 FB 13
BEGIN
   EN_R := TRUE;
   ID := W#16#16;
   R_ID := DW#16#16;
   NDR := FALSE;
   ERROR := FALSE;
   STATUS := W#16#0;
   RD_1 := P#DB28.DBX 0.0 BYTE 10;
   LEN := W#16#0;
   FB_ZUSTAND := B#16#0;
   EN_R_SAVE := FALSE;
   ID_SAVE := W#16#0;
   R_ID_SAVE := DW#16#0;
   FC_DATA_LEN := W#16#0;
   SD_1_SAVE0 := W#16#0;
   SD_1_SAVE2 := W#16#0;
   SD_1_SAVE4 := W#16#0;
   SD_1_SAVE6 := W#16#0;
   SD_1_SAVE8 := W#16#0;
   HS_REQ_BYTE.rii := FALSE;
   HS_REQ_BYTE.nva := FALSE;
   HS_REQ_BYTE.ofs := FALSE;
   HS_REQ_BYTE.dir := FALSE;
   HS_REQ_BYTE.res := FALSE;
   HS_REQ_BYTE.roc := FALSE;
   HS_REQ_BYTE.nls := FALSE;
   HS_REQ_BYTE.rlo := FALSE;
   HS_RESP_BYTE.aii := FALSE;
   HS_RESP_BYTE.sns := FALSE;
   HS_RESP_BYTE.sqc := FALSE;
   HS_RESP_BYTE.ads := FALSE;
   HS_RESP_BYTE.aoc := FALSE;
   HS_RESP_BYTE.rs1 := FALSE;
   HS_RESP_BYTE.cnr := FALSE;
   HS_RESP_BYTE.rs2 := FALSE;
   HS_RESP_DSNR := B#16#0;
   HS_RESP_OFFSET := W#16#0;
   SD_1_WORD0 := W#16#0;
   SD_1_COUNT := W#16#0;
   SD_1_DBNUMMER := W#16#0;
   SD_1_DWORD6 := DW#16#0;
   SD_1_TYP := B#16#0;
   SFC_PARAM.LEN := W#16#0;
   SFC_PARAM.DB_NUMMER := W#16#0;
   SFC_PARAM.START := DW#16#0;
   BUFFER[0] := W#16#0;
   BUFFER[1] := W#16#0;
   BUFFER[2] := W#16#0;
   BUFFER[3] := W#16#0;
   BUFFER[4] := W#16#0;
   BUFFER[5] := W#16#0;
   BUFFER[6] := W#16#0;
   BUFFER[7] := W#16#0;
   BUFFER[8] := W#16#0;
   BUFFER[9] := W#16#0;
   BUFFER[10] := W#16#0;
   BUFFER[11] := W#16#0;
   BUFFER[12] := W#16#0;
   BUFFER[13] := W#16#0;
   BUFFER[14] := W#16#0;
   BUFFER[15] := W#16#0;
   BUFFER[16] := W#16#0;
   BUFFER[17] := W#16#0;
   BUFFER[18] := W#16#0;
   BUFFER[19] := W#16#0;
   BUFFER[20] := W#16#0;
   BUFFER[21] := W#16#0;
   BUFFER[22] := W#16#0;
   BUFFER[23] := W#16#0;
   BUFFER[24] := W#16#0;
   BUFFER[25] := W#16#0;
   BUFFER[26] := W#16#0;
   BUFFER[27] := W#16#0;
   BUFFER[28] := W#16#0;
   BUFFER[29] := W#16#0;
   BUFFER[30] := W#16#0;
   BUFFER[31] := W#16#0;
   BUFFER[32] := W#16#0;
   BUFFER[33] := W#16#0;
   BUFFER[34] := W#16#0;
   BUFFER[35] := W#16#0;
   BUFFER[36] := W#16#0;
   BUFFER[37] := W#16#0;
   BUFFER[38] := W#16#0;
   BUFFER[39] := W#16#0;
   BUFFER[40] := W#16#0;
   BUFFER[41] := W#16#0;
   BUFFER[42] := W#16#0;
   BUFFER[43] := W#16#0;
   BUFFER[44] := W#16#0;
   BUFFER[45] := W#16#0;
   BUFFER[46] := W#16#0;
   BUFFER[47] := W#16#0;
   BUFFER[48] := W#16#0;
   BUFFER[49] := W#16#0;
   BUFFER[50] := W#16#0;
   BUFFER[51] := W#16#0;
   BUFFER[52] := W#16#0;
   BUFFER[53] := W#16#0;
   BUFFER[54] := W#16#0;
   BUFFER[55] := W#16#0;
   BUFFER[56] := W#16#0;
   BUFFER[57] := W#16#0;
   BUFFER[58] := W#16#0;
   BUFFER[59] := W#16#0;
   BUFFER[60] := W#16#0;
   BUFFER[61] := W#16#0;
   BUFFER[62] := W#16#0;
   BUFFER[63] := W#16#0;
   BUFFER[64] := W#16#0;
   BUFFER[65] := W#16#0;
   BUFFER[66] := W#16#0;
   BUFFER[67] := W#16#0;
   BUFFER[68] := W#16#0;
   BUFFER[69] := W#16#0;
   BUFFER[70] := W#16#0;
   BUFFER[71] := W#16#0;
   BUFFER[72] := W#16#0;
   BUFFER[73] := W#16#0;
   BUFFER[74] := W#16#0;
   BUFFER[75] := W#16#0;
   BUFFER[76] := W#16#0;
   BUFFER[77] := W#16#0;
   BUFFER[78] := W#16#0;
   BUFFER[79] := W#16#0;
   BUFFER[80] := W#16#0;
   BUFFER[81] := W#16#0;
   BUFFER[82] := W#16#0;
   BUFFER[83] := W#16#0;
   BUFFER[84] := W#16#0;
   BUFFER[85] := W#16#0;
   BUFFER[86] := W#16#0;
   BUFFER[87] := W#16#0;
   BUFFER[88] := W#16#0;
   BUFFER[89] := W#16#0;
   BUFFER[90] := W#16#0;
   BUFFER[91] := W#16#0;
   BUFFER[92] := W#16#0;
   BUFFER[93] := W#16#0;
   BUFFER[94] := W#16#0;
   BUFFER[95] := W#16#0;
   BUFFER[96] := W#16#0;
   BUFFER[97] := W#16#0;
   BUFFER[98] := W#16#0;
   BUFFER[99] := W#16#0;
   BUFFER[100] := W#16#0;
   BUFFER[101] := W#16#0;
   BUFFER[102] := W#16#0;
   BUFFER[103] := W#16#0;
   BUFFER[104] := W#16#0;
   BUFFER[105] := W#16#0;
   BUFFER[106] := W#16#0;
   BUFFER[107] := W#16#0;
   BUFFER[108] := W#16#0;
   BUFFER[109] := W#16#0;
   BUFFER[110] := W#16#0;
   BUFFER[111] := W#16#0;
   BUFFER[112] := W#16#0;
   BUFFER[113] := W#16#0;
   BUFFER[114] := W#16#0;
   BUFFER[115] := W#16#0;
   BUFFER[116] := W#16#0;
   BUFFER[117] := W#16#0;
   BUFFER[118] := W#16#0;
   BUFFER[119] := W#16#0;
   REASON_FOR_CLOSE := B#16#0;
   DS_NR := B#16#0;
   MAX_PUFF_LEN_SAVE := W#16#0;
   TYP_BOOL := FALSE;
   KANAL_PROBLEM := FALSE;
   KOMM_PROBLEM := FALSE;
   RECV_STARTED := FALSE;
   SEND_STARTED := FALSE;
   RESET_REQUEST := FALSE;
   RESET_EXECUTED := FALSE;
   DS200_BUSY := FALSE;
   LADDR_PTR := DW#16#0;
   LADDR := W#16#0;
   ZIEL_BYTE_SAVE := B#16#0;
   BOOL_ZIEL_BAD := FALSE;
   PARAM_OFFSET := DW#16#0;
   SLEEP := B#16#0;
   SLEEP_EXT := B#16#0;
   ID_CLOSE := W#16#0;
   RUNNING_LEN := W#16#0;
   FB_KENNUNG := B#16#F2;
   RESERVE := B#16#0;
   ZUSTAND_WEICHE := B#16#2;
   SFB_AUFRUF.EN_R := TRUE;
   SFB_AUFRUF.ID := W#16#16;
   SFB_AUFRUF.R_ID := DW#16#16;
   SFB_AUFRUF.NDR := FALSE;
   SFB_AUFRUF.ERROR := FALSE;
   SFB_AUFRUF.STATUS := W#16#0;
   SFB_AUFRUF.RD_1 := P#DB28.DBX 0.0 BYTE 10;
   SFB_AUFRUF.LEN := W#16#0;
   SFB_AUFRUF.INDEX := W#16#801;
   ZUSTAND_WEICHE_1 := B#16#CA;
END_DATA_BLOCK

DATA_BLOCK DB 326
TITLE =
AUTHOR : ICom
FAMILY : DIAGNOSE
VERSION : 0.0

 FB 327
BEGIN
   IN0 := 327;
   OUT1 := DW#16#0;
   STAT2[1] := B#16#0;
   STAT2[2] := B#16#64;
   STAT2[3] := B#16#1;
   STAT2[4] := B#16#10;
   STAT2[5] := B#16#F0;
   STAT2[6] := B#16#0;
   STAT2[7] := B#16#0;
   STAT2[8] := B#16#0;
   STAT2[9] := B#16#0;
   STAT2[10] := B#16#0;
   STAT2[11] := B#16#0;
   STAT2[12] := B#16#0;
   STAT2[13] := B#16#0;
   STAT2[14] := B#16#0;
   STAT2[15] := B#16#0;
   STAT2[16] := B#16#0;
   STAT2[17] := B#16#0;
   STAT2[18] := B#16#0;
   STAT2[19] := B#16#0;
   STAT2[20] := B#16#0;
   STAT2[21] := B#16#40;
   STAT2[22] := B#16#0;
   STAT2[23] := B#16#0;
   STAT2[24] := B#16#0;
   STAT2[25] := B#16#0;
   STAT2[26] := B#16#0;
   STAT2[27] := B#16#0;
   STAT2[28] := B#16#0;
   STAT2[29] := B#16#0;
   STAT2[30] := B#16#0;
   STAT2[31] := B#16#0;
   STAT2[32] := B#16#0;
   STAT2[33] := B#16#0;
   STAT2[34] := B#16#0;
   STAT2[35] := B#16#0;
   STAT2[36] := B#16#0;
   STAT2[37] := B#16#0;
   STAT2[38] := B#16#0;
   STAT2[39] := B#16#0;
   STAT2[40] := B#16#0;
   STAT2[41] := B#16#0;
   STAT2[42] := B#16#0;
   STAT2[43] := B#16#0;
   STAT2[44] := B#16#0;
   STAT2[45] := B#16#0;
   STAT2[46] := B#16#0;
   STAT2[47] := B#16#0;
   STAT2[48] := B#16#0;
   STAT2[49] := B#16#0;
   STAT2[50] := B#16#0;
   STAT2[51] := B#16#0;
   STAT2[52] := B#16#0;
   STAT2[53] := B#16#0;
   STAT2[54] := B#16#0;
   STAT2[55] := B#16#0;
   STAT2[56] := B#16#0;
   STAT2[57] := B#16#0;
   STAT2[58] := B#16#0;
   STAT2[59] := B#16#0;
   STAT2[60] := B#16#0;
   STAT2[61] := B#16#0;
   STAT2[62] := B#16#0;
   STAT2[63] := B#16#0;
   STAT2[64] := B#16#0;
   STAT2[65] := B#16#0;
   STAT2[66] := B#16#0;
   STAT2[67] := B#16#0;
   STAT2[68] := B#16#0;
   STAT2[69] := B#16#0;
   STAT2[70] := B#16#0;
   STAT2[71] := B#16#0;
   STAT2[72] := B#16#0;
   STAT2[73] := B#16#0;
   STAT2[74] := B#16#0;
   STAT2[75] := B#16#0;
   STAT2[76] := B#16#0;
   STAT2[77] := B#16#0;
   STAT2[78] := B#16#0;
   STAT2[79] := B#16#0;
   STAT2[80] := B#16#0;
   STAT2[81] := B#16#0;
   STAT2[82] := B#16#0;
   STAT2[83] := B#16#0;
   STAT2[84] := B#16#0;
   STAT2[85] := B#16#0;
   STAT2[86] := B#16#0;
   STAT2[87] := B#16#0;
   STAT2[88] := B#16#0;
   STAT2[89] := B#16#0;
   STAT2[90] := B#16#0;
   STAT2[91] := B#16#0;
   STAT2[92] := B#16#0;
   STAT2[93] := B#16#0;
   STAT2[94] := B#16#0;
   STAT2[95] := B#16#0;
   STAT2[96] := B#16#0;
   STAT2[97] := B#16#0;
   STAT2[98] := B#16#0;
   STAT2[99] := B#16#0;
   STAT2[100] := B#16#0;
   STAT2[101] := B#16#0;
   STAT2[102] := B#16#0;
   STAT2[103] := B#16#0;
   STAT2[104] := B#16#0;
   STAT2[105] := B#16#0;
   STAT2[106] := B#16#0;
   STAT2[107] := B#16#0;
   STAT2[108] := B#16#0;
   STAT2[109] := B#16#0;
   STAT2[110] := B#16#0;
   STAT2[111] := B#16#0;
   STAT2[112] := B#16#0;
   STAT2[113] := B#16#0;
   STAT2[114] := B#16#0;
   STAT2[115] := B#16#0;
   STAT2[116] := B#16#0;
   STAT2[117] := B#16#0;
   STAT2[118] := B#16#0;
   STAT2[119] := B#16#0;
   STAT2[120] := B#16#0;
   STAT2[121] := B#16#0;
   STAT2[122] := B#16#0;
   STAT2[123] := B#16#0;
   STAT2[124] := B#16#0;
   STAT2[125] := B#16#0;
   STAT2[126] := B#16#0;
   STAT2[127] := B#16#0;
   STAT2[128] := B#16#0;
   STAT2[129] := B#16#0;
   STAT2[130] := B#16#0;
   STAT2[131] := B#16#0;
   STAT2[132] := B#16#0;
   STAT2[133] := B#16#0;
   STAT2[134] := B#16#0;
   STAT2[135] := B#16#0;
   STAT2[136] := B#16#0;
   STAT2[137] := B#16#0;
   STAT2[138] := B#16#0;
   STAT2[139] := B#16#0;
   STAT2[140] := B#16#0;
   STAT2[141] := B#16#0;
   STAT2[142] := B#16#0;
   STAT2[143] := B#16#0;
   STAT2[144] := B#16#0;
   STAT2[145] := B#16#0;
   STAT2[146] := B#16#0;
   STAT2[147] := B#16#0;
   STAT2[148] := B#16#0;
   STAT2[149] := B#16#0;
   STAT2[150] := B#16#0;
   STAT2[151] := B#16#0;
   STAT2[152] := B#16#0;
   STAT2[153] := B#16#0;
   STAT2[154] := B#16#0;
   STAT2[155] := B#16#0;
   STAT2[156] := B#16#0;
   STAT2[157] := B#16#0;
   STAT2[158] := B#16#0;
   STAT2[159] := B#16#0;
   STAT2[160] := B#16#0;
   STAT2[161] := B#16#0;
   STAT2[162] := B#16#0;
   STAT2[163] := B#16#0;
   STAT2[164] := B#16#0;
   STAT2[165] := B#16#0;
   STAT2[166] := B#16#0;
   STAT2[167] := B#16#0;
   STAT2[168] := B#16#0;
   STAT2[169] := B#16#0;
   STAT2[170] := B#16#0;
   STAT2[171] := B#16#0;
   STAT2[172] := B#16#0;
   STAT2[173] := B#16#0;
   STAT2[174] := B#16#0;
   STAT2[175] := B#16#0;
   STAT2[176] := B#16#0;
   STAT2[177] := B#16#0;
   STAT2[178] := B#16#0;
   STAT2[179] := B#16#0;
   STAT2[180] := B#16#0;
   STAT2[181] := B#16#0;
   STAT2[182] := B#16#0;
   STAT2[183] := B#16#0;
   STAT2[184] := B#16#0;
   STAT2[185] := B#16#0;
   STAT2[186] := B#16#0;
   STAT2[187] := B#16#0;
   STAT2[188] := B#16#0;
   STAT2[189] := B#16#0;
   STAT2[190] := B#16#0;
   STAT2[191] := B#16#0;
   STAT2[192] := B#16#0;
   STAT2[193] := B#16#0;
   STAT2[194] := B#16#0;
   STAT2[195] := B#16#0;
   STAT2[196] := B#16#0;
   STAT2[197] := B#16#0;
   STAT2[198] := B#16#0;
   STAT2[199] := B#16#0;
   STAT2[200] := B#16#0;
   STAT2[201] := B#16#0;
   STAT2[202] := B#16#0;
   STAT2[203] := B#16#0;
   STAT2[204] := B#16#0;
   STAT2[205] := B#16#0;
   STAT2[206] := B#16#0;
   STAT2[207] := B#16#0;
   STAT2[208] := B#16#0;
   STAT2[209] := B#16#0;
   STAT2[210] := B#16#0;
   STAT2[211] := B#16#0;
   STAT2[212] := B#16#0;
   STAT2[213] := B#16#0;
   STAT2[214] := B#16#0;
   STAT2[215] := B#16#0;
   STAT2[216] := B#16#0;
   STAT2[217] := B#16#0;
   STAT2[218] := B#16#0;
   STAT2[219] := B#16#0;
   STAT2[220] := B#16#0;
   STAT2[221] := B#16#0;
   STAT2[222] := B#16#0;
   STAT2[223] := B#16#0;
   STAT2[224] := B#16#0;
   STAT2[225] := B#16#0;
   STAT2[226] := B#16#0;
   STAT2[227] := B#16#0;
   STAT2[228] := B#16#0;
   STAT2[229] := B#16#0;
   STAT2[230] := B#16#0;
   STAT2[231] := B#16#0;
   STAT2[232] := B#16#0;
   STAT2[233] := B#16#0;
   STAT2[234] := B#16#0;
   STAT2[235] := B#16#0;
   STAT2[236] := B#16#0;
   STAT2[237] := B#16#0;
   STAT2[238] := B#16#0;
   STAT2[239] := B#16#0;
   STAT2[240] := B#16#0;
   STAT2[241] := B#16#0;
   STAT2[242] := B#16#0;
   STAT2[243] := B#16#0;
   STAT2[244] := B#16#0;
   STAT2[245] := B#16#0;
   STAT2[246] := B#16#0;
   STAT2[247] := B#16#0;
   STAT2[248] := B#16#0;
   STAT2[249] := B#16#0;
   STAT2[250] := B#16#0;
   STAT2[251] := B#16#0;
   STAT2[252] := B#16#0;
   STAT2[253] := B#16#0;
   STAT2[254] := B#16#0;
   STAT2[255] := B#16#0;
   STAT2[256] := B#16#0;
   STAT2[257] := B#16#0;
   STAT2[258] := B#16#0;
   STAT2[259] := B#16#0;
   STAT2[260] := B#16#64;
   STAT2[261] := B#16#1;
   STAT2[262] := B#16#10;
   STAT2[263] := B#16#F0;
   STAT2[264] := B#16#0;
   STAT2[265] := B#16#0;
   STAT2[266] := B#16#0;
   STAT2[267] := B#16#0;
   STAT2[268] := B#16#0;
   STAT2[269] := B#16#0;
   STAT2[270] := B#16#0;
   STAT2[271] := B#16#0;
   STAT2[272] := B#16#0;
   STAT2[273] := B#16#0;
   STAT2[274] := B#16#0;
   STAT2[275] := B#16#0;
   STAT2[276] := B#16#0;
   STAT2[277] := B#16#0;
   STAT2[278] := B#16#0;
   STAT2[279] := B#16#40;
   STAT2[280] := B#16#0;
   STAT2[281] := B#16#0;
   STAT2[282] := B#16#0;
   STAT2[283] := B#16#0;
   STAT2[284] := B#16#0;
   STAT2[285] := B#16#0;
   STAT2[286] := B#16#0;
   STAT2[287] := B#16#0;
   STAT2[288] := B#16#0;
   STAT2[289] := B#16#0;
   STAT2[290] := B#16#0;
   STAT2[291] := B#16#0;
   STAT2[292] := B#16#0;
   STAT2[293] := B#16#0;
   STAT2[294] := B#16#0;
   STAT2[295] := B#16#0;
   STAT2[296] := B#16#0;
   STAT2[297] := B#16#0;
   STAT2[298] := B#16#0;
   STAT2[299] := B#16#0;
   STAT2[300] := B#16#0;
   STAT2[301] := B#16#0;
   STAT2[302] := B#16#0;
   STAT2[303] := B#16#0;
   STAT2[304] := B#16#0;
   STAT2[305] := B#16#0;
   STAT2[306] := B#16#0;
   STAT2[307] := B#16#0;
   STAT2[308] := B#16#0;
   STAT2[309] := B#16#0;
   STAT2[310] := B#16#0;
   STAT2[311] := B#16#0;
   STAT2[312] := B#16#0;
   STAT2[313] := B#16#0;
   STAT2[314] := B#16#0;
   STAT2[315] := B#16#0;
   STAT2[316] := B#16#0;
   STAT2[317] := B#16#0;
   STAT2[318] := B#16#0;
   STAT2[319] := B#16#0;
   STAT2[320] := B#16#0;
   STAT2[321] := B#16#0;
   STAT2[322] := B#16#0;
   STAT2[323] := B#16#0;
   STAT2[324] := B#16#0;
   STAT2[325] := B#16#0;
   STAT2[326] := B#16#0;
   STAT2[327] := B#16#0;
   STAT2[328] := B#16#0;
   STAT2[329] := B#16#0;
   STAT2[330] := B#16#0;
   STAT2[331] := B#16#0;
   STAT2[332] := B#16#0;
   STAT2[333] := B#16#0;
   STAT2[334] := B#16#0;
   STAT2[335] := B#16#0;
   STAT2[336] := B#16#0;
   STAT2[337] := B#16#0;
   STAT2[338] := B#16#0;
   STAT2[339] := B#16#0;
   STAT2[340] := B#16#0;
   STAT2[341] := B#16#0;
   STAT2[342] := B#16#0;
   STAT2[343] := B#16#0;
   STAT2[344] := B#16#0;
   STAT2[345] := B#16#0;
   STAT2[346] := B#16#0;
   STAT2[347] := B#16#0;
   STAT2[348] := B#16#0;
   STAT2[349] := B#16#0;
   STAT2[350] := B#16#0;
   STAT2[351] := B#16#0;
   STAT2[352] := B#16#0;
   STAT2[353] := B#16#0;
   STAT2[354] := B#16#0;
   STAT2[355] := B#16#0;
   STAT2[356] := B#16#0;
   STAT2[357] := B#16#0;
   STAT2[358] := B#16#0;
   STAT2[359] := B#16#0;
   STAT2[360] := B#16#0;
   STAT2[361] := B#16#0;
   STAT2[362] := B#16#0;
   STAT2[363] := B#16#0;
   STAT2[364] := B#16#0;
   STAT2[365] := B#16#0;
   STAT2[366] := B#16#0;
   STAT2[367] := B#16#0;
   STAT2[368] := B#16#0;
   STAT2[369] := B#16#0;
   STAT2[370] := B#16#0;
   STAT2[371] := B#16#0;
   STAT2[372] := B#16#0;
   STAT2[373] := B#16#0;
   STAT2[374] := B#16#0;
   STAT2[375] := B#16#0;
   STAT2[376] := B#16#0;
   STAT2[377] := B#16#0;
   STAT2[378] := B#16#0;
   STAT2[379] := B#16#0;
   STAT2[380] := B#16#0;
   STAT2[381] := B#16#0;
   STAT2[382] := B#16#0;
   STAT2[383] := B#16#0;
   STAT2[384] := B#16#0;
   STAT2[385] := B#16#0;
   STAT2[386] := B#16#0;
   STAT2[387] := B#16#0;
   STAT2[388] := B#16#0;
   STAT2[389] := B#16#0;
   STAT2[390] := B#16#0;
   STAT2[391] := B#16#0;
   STAT2[392] := B#16#0;
   STAT2[393] := B#16#0;
   STAT2[394] := B#16#0;
   STAT2[395] := B#16#0;
   STAT2[396] := B#16#0;
   STAT2[397] := B#16#0;
   STAT2[398] := B#16#0;
   STAT2[399] := B#16#0;
   STAT2[400] := B#16#0;
   STAT2[401] := B#16#0;
   STAT2[402] := B#16#0;
   STAT2[403] := B#16#0;
   STAT2[404] := B#16#0;
   STAT2[405] := B#16#0;
   STAT2[406] := B#16#0;
   STAT2[407] := B#16#0;
   STAT2[408] := B#16#0;
   STAT2[409] := B#16#0;
   STAT2[410] := B#16#0;
   STAT2[411] := B#16#0;
   STAT2[412] := B#16#0;
   STAT2[413] := B#16#0;
   STAT2[414] := B#16#0;
   STAT2[415] := B#16#0;
   STAT2[416] := B#16#0;
   STAT2[417] := B#16#0;
   STAT2[418] := B#16#0;
   STAT2[419] := B#16#0;
   STAT2[420] := B#16#0;
   STAT2[421] := B#16#0;
   STAT2[422] := B#16#0;
   STAT2[423] := B#16#0;
   STAT2[424] := B#16#0;
   STAT2[425] := B#16#0;
   STAT2[426] := B#16#0;
   STAT2[427] := B#16#0;
   STAT2[428] := B#16#0;
   STAT2[429] := B#16#0;
   STAT2[430] := B#16#0;
   STAT2[431] := B#16#0;
   STAT2[432] := B#16#0;
   STAT2[433] := B#16#0;
   STAT2[434] := B#16#0;
   STAT2[435] := B#16#0;
   STAT2[436] := B#16#0;
   STAT2[437] := B#16#0;
   STAT2[438] := B#16#0;
   STAT2[439] := B#16#0;
   STAT2[440] := B#16#0;
   STAT2[441] := B#16#0;
   STAT2[442] := B#16#0;
   STAT2[443] := B#16#0;
   STAT2[444] := B#16#0;
   STAT2[445] := B#16#0;
   STAT2[446] := B#16#0;
   STAT2[447] := B#16#0;
   STAT2[448] := B#16#0;
   STAT2[449] := B#16#0;
   STAT2[450] := B#16#0;
   STAT2[451] := B#16#0;
   STAT2[452] := B#16#0;
   STAT2[453] := B#16#0;
   STAT2[454] := B#16#0;
   STAT2[455] := B#16#0;
   STAT2[456] := B#16#0;
   STAT2[457] := B#16#0;
   STAT2[458] := B#16#0;
   STAT2[459] := B#16#0;
   STAT2[460] := B#16#0;
   STAT2[461] := B#16#0;
   STAT2[462] := B#16#0;
   STAT2[463] := B#16#0;
   STAT2[464] := B#16#0;
   STAT2[465] := B#16#0;
   STAT2[466] := B#16#0;
   STAT2[467] := B#16#0;
   STAT2[468] := B#16#0;
   STAT2[469] := B#16#0;
   STAT2[470] := B#16#0;
   STAT2[471] := B#16#0;
   STAT2[472] := B#16#0;
   STAT2[473] := B#16#0;
   STAT2[474] := B#16#0;
   STAT2[475] := B#16#0;
   STAT2[476] := B#16#0;
   STAT2[477] := B#16#0;
   STAT2[478] := B#16#0;
   STAT2[479] := B#16#0;
   STAT2[480] := B#16#0;
   STAT2[481] := B#16#0;
   STAT2[482] := B#16#0;
   STAT2[483] := B#16#0;
   STAT2[484] := B#16#0;
   STAT2[485] := B#16#0;
   STAT2[486] := B#16#0;
   STAT2[487] := B#16#0;
   STAT2[488] := B#16#0;
   STAT2[489] := B#16#0;
   STAT2[490] := B#16#0;
   STAT2[491] := B#16#0;
   STAT2[492] := B#16#0;
   STAT2[493] := B#16#0;
   STAT2[494] := B#16#0;
   STAT2[495] := B#16#0;
   STAT2[496] := B#16#0;
   STAT2[497] := B#16#0;
   STAT2[498] := B#16#0;
   STAT2[499] := B#16#0;
   STAT2[500] := B#16#0;
   STAT2[501] := B#16#0;
   STAT2[502] := B#16#0;
   STAT2[503] := B#16#0;
   STAT2[504] := B#16#0;
   STAT2[505] := B#16#0;
   STAT2[506] := B#16#0;
   STAT2[507] := B#16#0;
   STAT2[508] := B#16#0;
   STAT2[509] := B#16#0;
   STAT2[510] := B#16#0;
   STAT2[511] := B#16#0;
   STAT2[512] := B#16#0;
   STAT2[513] := B#16#0;
   STAT2[514] := B#16#0;
   STAT2[515] := B#16#0;
   STAT2[516] := B#16#0;
   STAT2[517] := B#16#0;
   STAT2[518] := B#16#64;
   STAT2[519] := B#16#0;
   STAT2[520] := B#16#0;
   STAT2[521] := B#16#0;
   STAT2[522] := B#16#0;
   STAT2[523] := B#16#0;
   STAT2[524] := B#16#0;
   STAT2[525] := B#16#0;
   STAT2[526] := B#16#0;
   STAT2[527] := B#16#0;
   STAT2[528] := B#16#0;
   STAT2[529] := B#16#0;
   STAT2[530] := B#16#0;
   STAT2[531] := B#16#0;
   STAT2[532] := B#16#0;
   STAT2[533] := B#16#0;
   STAT2[534] := B#16#0;
   STAT2[535] := B#16#0;
   STAT2[536] := B#16#0;
   STAT2[537] := B#16#0;
   STAT2[538] := B#16#0;
   STAT2[539] := B#16#0;
   STAT2[540] := B#16#0;
   STAT2[541] := B#16#0;
   STAT2[542] := B#16#0;
   STAT2[543] := B#16#0;
   STAT2[544] := B#16#0;
   STAT2[545] := B#16#0;
   STAT2[546] := B#16#0;
   STAT2[547] := B#16#0;
   STAT2[548] := B#16#0;
   STAT2[549] := B#16#0;
   STAT2[550] := B#16#0;
   STAT2[551] := B#16#0;
   STAT2[552] := B#16#0;
   STAT2[553] := B#16#0;
   STAT2[554] := B#16#0;
   STAT2[555] := B#16#0;
   STAT2[556] := B#16#0;
   STAT2[557] := B#16#0;
   STAT2[558] := B#16#0;
   STAT2[559] := B#16#0;
   STAT2[560] := B#16#0;
   STAT2[561] := B#16#0;
   STAT2[562] := B#16#0;
   STAT2[563] := B#16#0;
   STAT2[564] := B#16#0;
   STAT2[565] := B#16#0;
   STAT2[566] := B#16#0;
   STAT2[567] := B#16#0;
   STAT2[568] := B#16#0;
   STAT2[569] := B#16#0;
   STAT2[570] := B#16#0;
   STAT2[571] := B#16#0;
   STAT2[572] := B#16#0;
   STAT2[573] := B#16#0;
   STAT2[574] := B#16#0;
   STAT2[575] := B#16#0;
   STAT2[576] := B#16#0;
   STAT2[577] := B#16#0;
   STAT2[578] := B#16#0;
   STAT2[579] := B#16#0;
   STAT2[580] := B#16#0;
   STAT2[581] := B#16#0;
   STAT2[582] := B#16#0;
   STAT2[583] := B#16#0;
   STAT2[584] := B#16#0;
   STAT2[585] := B#16#0;
   STAT2[586] := B#16#0;
   STAT2[587] := B#16#0;
   STAT2[588] := B#16#0;
   STAT2[589] := B#16#0;
   STAT2[590] := B#16#0;
   STAT2[591] := B#16#0;
   STAT2[592] := B#16#0;
   STAT2[593] := B#16#0;
   STAT2[594] := B#16#0;
   STAT2[595] := B#16#0;
   STAT2[596] := B#16#0;
   STAT2[597] := B#16#0;
   STAT2[598] := B#16#0;
   STAT2[599] := B#16#0;
   STAT2[600] := B#16#0;
   STAT2[601] := B#16#0;
   STAT2[602] := B#16#0;
   STAT2[603] := B#16#0;
   STAT2[604] := B#16#0;
   STAT2[605] := B#16#0;
   STAT2[606] := B#16#0;
   STAT2[607] := B#16#0;
   STAT2[608] := B#16#0;
   STAT2[609] := B#16#0;
   STAT2[610] := B#16#0;
   STAT2[611] := B#16#0;
   STAT2[612] := B#16#0;
   STAT2[613] := B#16#0;
   STAT2[614] := B#16#0;
   STAT2[615] := B#16#0;
   STAT2[616] := B#16#0;
   STAT2[617] := B#16#0;
   STAT2[618] := B#16#0;
   STAT2[619] := B#16#0;
   STAT2[620] := B#16#0;
   STAT2[621] := B#16#0;
   STAT2[622] := B#16#0;
   STAT2[623] := B#16#0;
   STAT2[624] := B#16#0;
   STAT2[625] := B#16#0;
   STAT2[626] := B#16#0;
   STAT2[627] := B#16#0;
   STAT2[628] := B#16#0;
   STAT2[629] := B#16#0;
   STAT2[630] := B#16#0;
   STAT2[631] := B#16#0;
   STAT2[632] := B#16#0;
   STAT2[633] := B#16#0;
   STAT2[634] := B#16#0;
   STAT2[635] := B#16#0;
   STAT2[636] := B#16#0;
   STAT2[637] := B#16#0;
   STAT2[638] := B#16#0;
   STAT2[639] := B#16#0;
   STAT2[640] := B#16#0;
   STAT2[641] := B#16#0;
   STAT2[642] := B#16#0;
   STAT2[643] := B#16#0;
   STAT2[644] := B#16#0;
   STAT2[645] := B#16#0;
   STAT2[646] := B#16#0;
   STAT2[647] := B#16#0;
   STAT2[648] := B#16#0;
   STAT2[649] := B#16#0;
   STAT2[650] := B#16#0;
   STAT2[651] := B#16#0;
   STAT2[652] := B#16#0;
   STAT2[653] := B#16#0;
   STAT2[654] := B#16#0;
   STAT2[655] := B#16#0;
   STAT2[656] := B#16#0;
   STAT2[657] := B#16#0;
   STAT2[658] := B#16#0;
   STAT2[659] := B#16#0;
   STAT2[660] := B#16#0;
   STAT2[661] := B#16#0;
   STAT2[662] := B#16#0;
   STAT2[663] := B#16#0;
   STAT2[664] := B#16#0;
   STAT2[665] := B#16#0;
   STAT2[666] := B#16#0;
   STAT2[667] := B#16#0;
   STAT2[668] := B#16#0;
   STAT2[669] := B#16#0;
   STAT2[670] := B#16#0;
   STAT2[671] := B#16#0;
   STAT2[672] := B#16#0;
   STAT2[673] := B#16#0;
   STAT2[674] := B#16#0;
   STAT2[675] := B#16#0;
   STAT2[676] := B#16#0;
   STAT2[677] := B#16#0;
   STAT2[678] := B#16#0;
   STAT2[679] := B#16#0;
   STAT2[680] := B#16#0;
   STAT2[681] := B#16#0;
   STAT2[682] := B#16#0;
   STAT2[683] := B#16#0;
   STAT2[684] := B#16#0;
   STAT2[685] := B#16#0;
   STAT2[686] := B#16#0;
   STAT2[687] := B#16#0;
   STAT2[688] := B#16#0;
   STAT2[689] := B#16#0;
   STAT2[690] := B#16#0;
   STAT2[691] := B#16#0;
   STAT2[692] := B#16#0;
   STAT2[693] := B#16#0;
   STAT2[694] := B#16#0;
   STAT2[695] := B#16#0;
   STAT2[696] := B#16#0;
   STAT2[697] := B#16#0;
   STAT2[698] := B#16#0;
   STAT2[699] := B#16#0;
   STAT2[700] := B#16#0;
   STAT2[701] := B#16#0;
   STAT2[702] := B#16#0;
   STAT2[703] := B#16#0;
   STAT2[704] := B#16#0;
   STAT2[705] := B#16#0;
   STAT2[706] := B#16#0;
   STAT2[707] := B#16#0;
   STAT2[708] := B#16#0;
   STAT2[709] := B#16#0;
   STAT2[710] := B#16#0;
   STAT2[711] := B#16#0;
   STAT2[712] := B#16#0;
   STAT2[713] := B#16#0;
   STAT2[714] := B#16#0;
   STAT2[715] := B#16#0;
   STAT2[716] := B#16#0;
   STAT2[717] := B#16#0;
   STAT2[718] := B#16#0;
   STAT2[719] := B#16#0;
   STAT2[720] := B#16#0;
   STAT2[721] := B#16#0;
   STAT2[722] := B#16#0;
   STAT2[723] := B#16#0;
   STAT2[724] := B#16#0;
   STAT2[725] := B#16#0;
   STAT2[726] := B#16#0;
   STAT2[727] := B#16#0;
   STAT2[728] := B#16#0;
   STAT2[729] := B#16#0;
   STAT2[730] := B#16#0;
   STAT2[731] := B#16#0;
   STAT2[732] := B#16#0;
   STAT2[733] := B#16#0;
   STAT2[734] := B#16#0;
   STAT2[735] := B#16#0;
   STAT2[736] := B#16#0;
   STAT2[737] := B#16#0;
   STAT2[738] := B#16#0;
   STAT2[739] := B#16#0;
   STAT2[740] := B#16#0;
   STAT2[741] := B#16#0;
   STAT2[742] := B#16#0;
   STAT2[743] := B#16#0;
   STAT2[744] := B#16#0;
   STAT2[745] := B#16#0;
   STAT2[746] := B#16#0;
   STAT2[747] := B#16#0;
   STAT2[748] := B#16#0;
   STAT2[749] := B#16#0;
   STAT2[750] := B#16#0;
   STAT2[751] := B#16#0;
   STAT2[752] := B#16#0;
   STAT2[753] := B#16#0;
   STAT2[754] := B#16#0;
   STAT2[755] := B#16#0;
   STAT2[756] := B#16#0;
   STAT2[757] := B#16#0;
   STAT2[758] := B#16#0;
   STAT2[759] := B#16#0;
   STAT2[760] := B#16#0;
   STAT2[761] := B#16#0;
   STAT2[762] := B#16#0;
   STAT2[763] := B#16#0;
   STAT2[764] := B#16#0;
   STAT2[765] := B#16#0;
   STAT2[766] := B#16#0;
   STAT2[767] := B#16#0;
   STAT2[768] := B#16#0;
   STAT2[769] := B#16#0;
   STAT2[770] := B#16#0;
   STAT2[771] := B#16#0;
   STAT2[772] := B#16#0;
   STAT2[773] := B#16#0;
   STAT2[774] := B#16#0;
   STAT2[775] := B#16#0;
   STAT2[776] := B#16#64;
   STAT2[777] := B#16#0;
   STAT2[778] := B#16#0;
   STAT2[779] := B#16#0;
   STAT2[780] := B#16#0;
   STAT2[781] := B#16#0;
   STAT2[782] := B#16#0;
   STAT2[783] := B#16#0;
   STAT2[784] := B#16#0;
   STAT2[785] := B#16#0;
   STAT2[786] := B#16#0;
   STAT2[787] := B#16#0;
   STAT2[788] := B#16#0;
   STAT2[789] := B#16#0;
   STAT2[790] := B#16#0;
   STAT2[791] := B#16#0;
   STAT2[792] := B#16#0;
   STAT2[793] := B#16#0;
   STAT2[794] := B#16#0;
   STAT2[795] := B#16#0;
   STAT2[796] := B#16#0;
   STAT2[797] := B#16#0;
   STAT2[798] := B#16#0;
   STAT2[799] := B#16#0;
   STAT2[800] := B#16#0;
   STAT2[801] := B#16#0;
   STAT2[802] := B#16#0;
   STAT2[803] := B#16#0;
   STAT2[804] := B#16#0;
   STAT2[805] := B#16#0;
   STAT2[806] := B#16#0;
   STAT2[807] := B#16#0;
   STAT2[808] := B#16#0;
   STAT2[809] := B#16#0;
   STAT2[810] := B#16#0;
   STAT2[811] := B#16#0;
   STAT2[812] := B#16#0;
   STAT2[813] := B#16#0;
   STAT2[814] := B#16#0;
   STAT2[815] := B#16#0;
   STAT2[816] := B#16#0;
   STAT2[817] := B#16#0;
   STAT2[818] := B#16#0;
   STAT2[819] := B#16#0;
   STAT2[820] := B#16#0;
   STAT2[821] := B#16#0;
   STAT2[822] := B#16#0;
   STAT2[823] := B#16#0;
   STAT2[824] := B#16#0;
   STAT2[825] := B#16#0;
   STAT2[826] := B#16#0;
   STAT2[827] := B#16#0;
   STAT2[828] := B#16#0;
   STAT2[829] := B#16#0;
   STAT2[830] := B#16#0;
   STAT2[831] := B#16#0;
   STAT2[832] := B#16#0;
   STAT2[833] := B#16#0;
   STAT2[834] := B#16#0;
   STAT2[835] := B#16#0;
   STAT2[836] := B#16#0;
   STAT2[837] := B#16#0;
   STAT2[838] := B#16#0;
   STAT2[839] := B#16#0;
   STAT2[840] := B#16#0;
   STAT2[841] := B#16#0;
   STAT2[842] := B#16#0;
   STAT2[843] := B#16#0;
   STAT2[844] := B#16#0;
   STAT2[845] := B#16#0;
   STAT2[846] := B#16#0;
   STAT2[847] := B#16#0;
   STAT2[848] := B#16#0;
   STAT2[849] := B#16#0;
   STAT2[850] := B#16#0;
   STAT2[851] := B#16#0;
   STAT2[852] := B#16#0;
   STAT2[853] := B#16#0;
   STAT2[854] := B#16#0;
   STAT2[855] := B#16#0;
   STAT2[856] := B#16#0;
   STAT2[857] := B#16#0;
   STAT2[858] := B#16#0;
   STAT2[859] := B#16#0;
   STAT2[860] := B#16#0;
   STAT2[861] := B#16#0;
   STAT2[862] := B#16#0;
   STAT2[863] := B#16#0;
   STAT2[864] := B#16#0;
   STAT2[865] := B#16#0;
   STAT2[866] := B#16#0;
   STAT2[867] := B#16#0;
   STAT2[868] := B#16#0;
   STAT2[869] := B#16#0;
   STAT2[870] := B#16#0;
   STAT2[871] := B#16#0;
   STAT2[872] := B#16#0;
   STAT2[873] := B#16#0;
   STAT2[874] := B#16#0;
   STAT2[875] := B#16#0;
   STAT2[876] := B#16#0;
   STAT2[877] := B#16#0;
   STAT2[878] := B#16#0;
   STAT2[879] := B#16#0;
   STAT2[880] := B#16#0;
   STAT2[881] := B#16#0;
   STAT2[882] := B#16#0;
   STAT2[883] := B#16#0;
   STAT2[884] := B#16#0;
   STAT2[885] := B#16#0;
   STAT2[886] := B#16#0;
   STAT2[887] := B#16#0;
   STAT2[888] := B#16#0;
   STAT2[889] := B#16#0;
   STAT2[890] := B#16#0;
   STAT2[891] := B#16#0;
   STAT2[892] := B#16#0;
   STAT2[893] := B#16#0;
   STAT2[894] := B#16#0;
   STAT2[895] := B#16#0;
   STAT2[896] := B#16#0;
   STAT2[897] := B#16#0;
   STAT2[898] := B#16#0;
   STAT2[899] := B#16#0;
   STAT2[900] := B#16#0;
   STAT2[901] := B#16#0;
   STAT2[902] := B#16#0;
   STAT2[903] := B#16#0;
   STAT2[904] := B#16#0;
   STAT2[905] := B#16#0;
   STAT2[906] := B#16#0;
   STAT2[907] := B#16#0;
   STAT2[908] := B#16#0;
   STAT2[909] := B#16#0;
   STAT2[910] := B#16#0;
   STAT2[911] := B#16#0;
   STAT2[912] := B#16#0;
   STAT2[913] := B#16#0;
   STAT2[914] := B#16#0;
   STAT2[915] := B#16#0;
   STAT2[916] := B#16#0;
   STAT2[917] := B#16#0;
   STAT2[918] := B#16#0;
   STAT2[919] := B#16#0;
   STAT2[920] := B#16#0;
   STAT2[921] := B#16#0;
   STAT2[922] := B#16#0;
   STAT2[923] := B#16#0;
   STAT2[924] := B#16#0;
   STAT2[925] := B#16#0;
   STAT2[926] := B#16#0;
   STAT2[927] := B#16#0;
   STAT2[928] := B#16#0;
   STAT2[929] := B#16#0;
   STAT2[930] := B#16#0;
   STAT2[931] := B#16#0;
   STAT2[932] := B#16#0;
   STAT2[933] := B#16#0;
   STAT2[934] := B#16#0;
   STAT2[935] := B#16#0;
   STAT2[936] := B#16#0;
   STAT2[937] := B#16#0;
   STAT2[938] := B#16#0;
   STAT2[939] := B#16#0;
   STAT2[940] := B#16#0;
   STAT2[941] := B#16#0;
   STAT2[942] := B#16#0;
   STAT2[943] := B#16#0;
   STAT2[944] := B#16#0;
   STAT2[945] := B#16#0;
   STAT2[946] := B#16#0;
   STAT2[947] := B#16#0;
   STAT2[948] := B#16#0;
   STAT2[949] := B#16#0;
   STAT2[950] := B#16#0;
   STAT2[951] := B#16#0;
   STAT2[952] := B#16#0;
   STAT2[953] := B#16#0;
   STAT2[954] := B#16#0;
   STAT2[955] := B#16#0;
   STAT2[956] := B#16#0;
   STAT2[957] := B#16#0;
   STAT2[958] := B#16#0;
   STAT2[959] := B#16#0;
   STAT2[960] := B#16#0;
   STAT2[961] := B#16#0;
   STAT2[962] := B#16#0;
   STAT2[963] := B#16#0;
   STAT2[964] := B#16#0;
   STAT2[965] := B#16#0;
   STAT2[966] := B#16#0;
   STAT2[967] := B#16#0;
   STAT2[968] := B#16#0;
   STAT2[969] := B#16#0;
   STAT2[970] := B#16#0;
   STAT2[971] := B#16#0;
   STAT2[972] := B#16#0;
   STAT2[973] := B#16#0;
   STAT2[974] := B#16#0;
   STAT2[975] := B#16#0;
   STAT2[976] := B#16#0;
   STAT2[977] := B#16#0;
   STAT2[978] := B#16#0;
   STAT2[979] := B#16#0;
   STAT2[980] := B#16#0;
   STAT2[981] := B#16#0;
   STAT2[982] := B#16#0;
   STAT2[983] := B#16#0;
   STAT2[984] := B#16#0;
   STAT2[985] := B#16#0;
   STAT2[986] := B#16#0;
   STAT2[987] := B#16#0;
   STAT2[988] := B#16#0;
   STAT2[989] := B#16#0;
   STAT2[990] := B#16#0;
   STAT2[991] := B#16#0;
   STAT2[992] := B#16#0;
   STAT2[993] := B#16#0;
   STAT2[994] := B#16#0;
   STAT2[995] := B#16#0;
   STAT2[996] := B#16#0;
   STAT2[997] := B#16#0;
   STAT2[998] := B#16#0;
   STAT2[999] := B#16#0;
   STAT2[1000] := B#16#0;
   STAT2[1001] := B#16#0;
   STAT2[1002] := B#16#0;
   STAT2[1003] := B#16#0;
   STAT2[1004] := B#16#0;
   STAT2[1005] := B#16#0;
   STAT2[1006] := B#16#0;
   STAT2[1007] := B#16#0;
   STAT2[1008] := B#16#0;
   STAT2[1009] := B#16#0;
   STAT2[1010] := B#16#0;
   STAT2[1011] := B#16#0;
   STAT2[1012] := B#16#0;
   STAT2[1013] := B#16#0;
   STAT2[1014] := B#16#0;
   STAT2[1015] := B#16#0;
   STAT2[1016] := B#16#0;
   STAT2[1017] := B#16#0;
   STAT2[1018] := B#16#0;
   STAT2[1019] := B#16#0;
   STAT2[1020] := B#16#0;
   STAT2[1021] := B#16#0;
   STAT2[1022] := B#16#0;
   STAT2[1023] := B#16#0;
   STAT2[1024] := B#16#0;
   STAT2[1025] := B#16#0;
   STAT2[1026] := B#16#0;
   STAT2[1027] := B#16#0;
   STAT2[1028] := B#16#0;
   STAT2[1029] := B#16#0;
   STAT2[1030] := B#16#0;
   STAT2[1031] := B#16#0;
   STAT2[1032] := B#16#0;
   STAT3[1] := B#16#0;
   STAT3[2] := B#16#0;
   STAT3[3] := B#16#0;
   STAT3[4] := B#16#0;
   STAT3[5] := B#16#0;
   STAT3[6] := B#16#0;
   STAT3[7] := B#16#0;
   STAT3[8] := B#16#0;
   STAT3[9] := B#16#0;
   STAT3[10] := B#16#0;
   STAT3[11] := B#16#0;
   STAT3[12] := B#16#0;
   STAT3[13] := B#16#0;
   STAT3[14] := B#16#0;
   STAT3[15] := B#16#0;
   STAT3[16] := B#16#0;
   STAT3[17] := B#16#0;
   STAT3[18] := B#16#0;
   STAT3[19] := B#16#0;
   STAT3[20] := B#16#0;
   STAT3[21] := B#16#0;
   STAT3[22] := B#16#0;
   STAT3[23] := B#16#0;
   STAT3[24] := B#16#1;
   STAT3[25] := B#16#0;
   STAT3[26] := B#16#0;
   STAT3[27] := B#16#0;
   STAT3[28] := B#16#0;
   STAT3[29] := B#16#0;
   STAT3[30] := B#16#0;
   STAT3[31] := B#16#0;
   STAT3[32] := B#16#0;
   STAT3[33] := B#16#0;
   STAT3[34] := B#16#0;
   STAT3[35] := B#16#0;
   STAT3[36] := B#16#0;
   STAT3[37] := B#16#0;
   STAT3[38] := B#16#0;
   STAT3[39] := B#16#0;
   STAT3[40] := B#16#1;
   STAT3[41] := B#16#0;
   STAT3[42] := B#16#1;
   STAT3[43] := B#16#0;
   STAT3[44] := B#16#1;
   STAT3[45] := B#16#0;
   STAT3[46] := B#16#1;
   STAT3[47] := B#16#0;
   STAT3[48] := B#16#0;
   STAT3[49] := B#16#0;
   STAT3[50] := B#16#0;
   STAT3[51] := B#16#0;
   STAT3[52] := B#16#0;
   STAT3[53] := B#16#0;
   STAT3[54] := B#16#0;
   STAT3[55] := B#16#0;
   STAT3[56] := B#16#0;
   STAT3[57] := B#16#0;
   STAT3[58] := B#16#0;
   STAT3[59] := B#16#0;
   STAT3[60] := B#16#0;
   STAT3[61] := B#16#0;
   STAT3[62] := B#16#0;
   STAT3[63] := B#16#0;
   STAT3[64] := B#16#0;
   STAT3[65] := B#16#0;
   STAT3[66] := B#16#0;
   STAT3[67] := B#16#0;
   STAT3[68] := B#16#0;
   STAT3[69] := B#16#0;
   STAT3[70] := B#16#0;
   STAT3[71] := B#16#0;
   STAT3[72] := B#16#0;
   STAT3[73] := B#16#0;
   STAT3[74] := B#16#0;
   STAT3[75] := B#16#0;
   STAT3[76] := B#16#0;
   STAT3[77] := B#16#0;
   STAT3[78] := B#16#0;
   STAT3[79] := B#16#0;
   STAT3[80] := B#16#0;
   STAT3[81] := B#16#0;
   STAT3[82] := B#16#0;
   STAT3[83] := B#16#0;
   STAT3[84] := B#16#0;
   STAT3[85] := B#16#0;
   STAT3[86] := B#16#0;
   STAT3[87] := B#16#0;
   STAT3[88] := B#16#0;
   STAT3[89] := B#16#0;
   STAT3[90] := B#16#0;
   STAT3[91] := B#16#0;
   STAT3[92] := B#16#0;
   STAT3[93] := B#16#0;
   STAT3[94] := B#16#0;
   STAT3[95] := B#16#0;
   STAT3[96] := B#16#0;
   STAT3[97] := B#16#0;
   STAT3[98] := B#16#0;
   STAT3[99] := B#16#0;
   STAT3[100] := B#16#0;
   STAT3[101] := B#16#0;
   STAT3[102] := B#16#0;
   STAT3[103] := B#16#0;
   STAT3[104] := B#16#0;
   STAT3[105] := B#16#0;
   STAT3[106] := B#16#0;
   STAT3[107] := B#16#0;
   STAT3[108] := B#16#0;
   STAT3[109] := B#16#0;
   STAT3[110] := B#16#0;
   STAT3[111] := B#16#0;
   STAT3[112] := B#16#0;
   STAT3[113] := B#16#0;
   STAT3[114] := B#16#0;
   STAT3[115] := B#16#0;
   STAT3[116] := B#16#0;
   STAT3[117] := B#16#0;
   STAT3[118] := B#16#0;
   STAT3[119] := B#16#0;
   STAT3[120] := B#16#0;
   STAT3[121] := B#16#0;
   STAT3[122] := B#16#0;
   STAT3[123] := B#16#0;
   STAT3[124] := B#16#0;
   STAT3[125] := B#16#0;
   STAT3[126] := B#16#0;
   STAT3[127] := B#16#0;
   STAT3[128] := B#16#0;
   STAT3[129] := B#16#0;
   STAT3[130] := B#16#0;
   STAT3[131] := B#16#0;
   STAT3[132] := B#16#0;
   STAT3[133] := B#16#0;
   STAT3[134] := B#16#0;
   STAT3[135] := B#16#0;
   STAT3[136] := B#16#0;
   STAT3[137] := B#16#0;
   STAT3[138] := B#16#0;
   STAT3[139] := B#16#0;
   STAT3[140] := B#16#0;
   STAT3[141] := B#16#0;
   STAT3[142] := B#16#0;
   STAT3[143] := B#16#0;
   STAT3[144] := B#16#0;
   STAT3[145] := B#16#0;
   STAT3[146] := B#16#0;
   STAT3[147] := B#16#0;
   STAT3[148] := B#16#0;
   STAT3[149] := B#16#0;
   STAT3[150] := B#16#0;
   STAT3[151] := B#16#0;
   STAT3[152] := B#16#0;
   STAT3[153] := B#16#0;
   STAT3[154] := B#16#0;
   STAT3[155] := B#16#0;
   STAT3[156] := B#16#0;
   STAT3[157] := B#16#0;
   STAT3[158] := B#16#0;
   STAT3[159] := B#16#0;
   STAT3[160] := B#16#0;
   STAT3[161] := B#16#0;
   STAT3[162] := B#16#0;
   STAT3[163] := B#16#0;
   STAT3[164] := B#16#0;
   STAT3[165] := B#16#0;
   STAT3[166] := B#16#0;
   STAT3[167] := B#16#0;
   STAT3[168] := B#16#0;
   STAT3[169] := B#16#0;
   STAT3[170] := B#16#0;
   STAT3[171] := B#16#0;
   STAT3[172] := B#16#0;
   STAT3[173] := B#16#0;
   STAT3[174] := B#16#0;
   STAT3[175] := B#16#0;
   STAT3[176] := B#16#0;
   STAT3[177] := B#16#0;
   STAT3[178] := B#16#0;
   STAT3[179] := B#16#0;
   STAT3[180] := B#16#0;
   STAT3[181] := B#16#0;
   STAT3[182] := B#16#0;
   STAT3[183] := B#16#0;
   STAT3[184] := B#16#0;
   STAT3[185] := B#16#0;
   STAT3[186] := B#16#0;
   STAT3[187] := B#16#0;
   STAT3[188] := B#16#0;
   STAT3[189] := B#16#0;
   STAT3[190] := B#16#0;
   STAT3[191] := B#16#0;
   STAT3[192] := B#16#0;
   STAT3[193] := B#16#0;
   STAT3[194] := B#16#0;
   STAT3[195] := B#16#0;
   STAT3[196] := B#16#0;
   STAT3[197] := B#16#0;
   STAT3[198] := B#16#0;
   STAT3[199] := B#16#0;
   STAT3[200] := B#16#0;
   STAT3[201] := B#16#0;
   STAT3[202] := B#16#0;
   STAT3[203] := B#16#0;
   STAT3[204] := B#16#0;
   STAT3[205] := B#16#0;
   STAT3[206] := B#16#0;
   STAT3[207] := B#16#0;
   STAT3[208] := B#16#0;
   STAT3[209] := B#16#0;
   STAT3[210] := B#16#0;
   STAT3[211] := B#16#0;
   STAT3[212] := B#16#0;
   STAT3[213] := B#16#0;
   STAT3[214] := B#16#0;
   STAT3[215] := B#16#0;
   STAT3[216] := B#16#0;
   STAT3[217] := B#16#0;
   STAT3[218] := B#16#0;
   STAT3[219] := B#16#0;
   STAT3[220] := B#16#0;
   STAT3[221] := B#16#0;
   STAT3[222] := B#16#0;
   STAT3[223] := B#16#0;
   STAT3[224] := B#16#0;
   STAT3[225] := B#16#0;
   STAT3[226] := B#16#0;
   STAT3[227] := B#16#0;
   STAT3[228] := B#16#0;
   STAT3[229] := B#16#0;
   STAT3[230] := B#16#0;
   STAT3[231] := B#16#0;
   STAT3[232] := B#16#0;
   STAT3[233] := B#16#0;
   STAT3[234] := B#16#0;
   STAT3[235] := B#16#0;
   STAT3[236] := B#16#0;
   STAT3[237] := B#16#0;
   STAT3[238] := B#16#0;
   STAT3[239] := B#16#0;
   STAT3[240] := B#16#0;
   STAT3[241] := B#16#0;
   STAT3[242] := B#16#0;
   STAT3[243] := B#16#0;
   STAT3[244] := B#16#0;
   STAT3[245] := B#16#0;
   STAT3[246] := B#16#0;
   STAT3[247] := B#16#0;
   STAT3[248] := B#16#0;
   STAT3[249] := B#16#0;
   STAT3[250] := B#16#0;
   STAT3[251] := B#16#0;
   STAT3[252] := B#16#0;
   STAT3[253] := B#16#0;
   STAT3[254] := B#16#0;
   STAT3[255] := B#16#0;
   STAT3[256] := B#16#0;
   STAT3[257] := B#16#0;
   STAT3[258] := B#16#0;
   STAT3[259] := B#16#0;
   STAT3[260] := B#16#0;
   STAT3[261] := B#16#0;
   STAT3[262] := B#16#0;
   STAT3[263] := B#16#0;
   STAT3[264] := B#16#0;
   STAT3[265] := B#16#0;
   STAT3[266] := B#16#0;
   STAT3[267] := B#16#0;
   STAT3[268] := B#16#0;
   STAT3[269] := B#16#0;
   STAT3[270] := B#16#0;
   STAT3[271] := B#16#0;
   STAT3[272] := B#16#0;
   STAT3[273] := B#16#0;
   STAT3[274] := B#16#0;
   STAT3[275] := B#16#0;
   STAT3[276] := B#16#0;
   STAT3[277] := B#16#0;
   STAT3[278] := B#16#0;
   STAT3[279] := B#16#0;
   STAT3[280] := B#16#0;
   STAT3[281] := B#16#0;
   STAT3[282] := B#16#0;
   STAT3[283] := B#16#0;
   STAT3[284] := B#16#0;
   STAT3[285] := B#16#0;
   STAT3[286] := B#16#0;
   STAT3[287] := B#16#0;
   STAT3[288] := B#16#0;
   STAT3[289] := B#16#0;
   STAT3[290] := B#16#0;
   STAT3[291] := B#16#0;
   STAT3[292] := B#16#0;
   STAT3[293] := B#16#0;
   STAT3[294] := B#16#0;
   STAT3[295] := B#16#0;
   STAT3[296] := B#16#0;
   STAT3[297] := B#16#0;
   STAT3[298] := B#16#0;
   STAT3[299] := B#16#0;
   STAT3[300] := B#16#1;
   STAT3[301] := B#16#0;
   STAT3[302] := B#16#0;
   STAT3[303] := B#16#0;
   STAT3[304] := B#16#0;
   STAT3[305] := B#16#0;
   STAT3[306] := B#16#0;
   STAT3[307] := B#16#0;
   STAT3[308] := B#16#0;
   STAT3[309] := B#16#0;
   STAT3[310] := B#16#0;
   STAT3[311] := B#16#0;
   STAT3[312] := B#16#0;
   STAT3[313] := B#16#0;
   STAT3[314] := B#16#0;
   STAT3[315] := B#16#0;
   STAT3[316] := B#16#0;
   STAT3[317] := B#16#0;
   STAT3[318] := B#16#0;
   STAT3[319] := B#16#0;
   STAT3[320] := B#16#0;
   STAT3[321] := B#16#0;
   STAT3[322] := B#16#0;
   STAT3[323] := B#16#0;
   STAT3[324] := B#16#0;
   STAT3[325] := B#16#0;
   STAT3[326] := B#16#0;
   STAT3[327] := B#16#0;
   STAT3[328] := B#16#0;
   STAT3[329] := B#16#0;
   STAT3[330] := B#16#0;
   STAT3[331] := B#16#0;
   STAT3[332] := B#16#0;
   STAT3[333] := B#16#0;
   STAT3[334] := B#16#0;
   STAT3[335] := B#16#0;
   STAT3[336] := B#16#0;
   STAT3[337] := B#16#0;
   STAT3[338] := B#16#0;
   STAT3[339] := B#16#0;
   STAT3[340] := B#16#0;
   STAT3[341] := B#16#0;
   STAT3[342] := B#16#0;
   STAT3[343] := B#16#0;
   STAT3[344] := B#16#0;
   STAT3[345] := B#16#0;
   STAT3[346] := B#16#0;
   STAT3[347] := B#16#0;
   STAT3[348] := B#16#0;
   STAT3[349] := B#16#0;
   STAT3[350] := B#16#0;
   STAT3[351] := B#16#0;
   STAT3[352] := B#16#0;
   STAT3[353] := B#16#0;
   STAT3[354] := B#16#0;
   STAT3[355] := B#16#0;
   STAT3[356] := B#16#0;
   STAT3[357] := B#16#0;
   STAT3[358] := B#16#0;
   STAT3[359] := B#16#0;
   STAT3[360] := B#16#0;
   STAT3[361] := B#16#0;
   STAT3[362] := B#16#0;
   STAT3[363] := B#16#0;
   STAT3[364] := B#16#0;
   STAT3[365] := B#16#0;
   STAT3[366] := B#16#0;
   STAT3[367] := B#16#0;
   STAT3[368] := B#16#0;
   STAT3[369] := B#16#0;
   STAT3[370] := B#16#0;
   STAT3[371] := B#16#0;
   STAT3[372] := B#16#0;
   STAT3[373] := B#16#0;
   STAT3[374] := B#16#0;
   STAT3[375] := B#16#0;
   STAT3[376] := B#16#0;
   STAT3[377] := B#16#0;
   STAT3[378] := B#16#0;
   STAT3[379] := B#16#0;
   STAT3[380] := B#16#0;
   STAT3[381] := B#16#0;
   STAT3[382] := B#16#0;
   STAT3[383] := B#16#0;
   STAT3[384] := B#16#0;
   STAT3[385] := B#16#0;
   STAT3[386] := B#16#0;
   STAT3[387] := B#16#0;
   STAT3[388] := B#16#0;
   STAT3[389] := B#16#0;
   STAT3[390] := B#16#0;
   STAT3[391] := B#16#0;
   STAT3[392] := B#16#0;
   STAT3[393] := B#16#0;
   STAT3[394] := B#16#0;
   STAT3[395] := B#16#0;
   STAT3[396] := B#16#0;
   STAT3[397] := B#16#0;
   STAT3[398] := B#16#0;
   STAT3[399] := B#16#0;
   STAT3[400] := B#16#0;
   STAT3[401] := B#16#0;
   STAT3[402] := B#16#0;
   STAT3[403] := B#16#0;
   STAT3[404] := B#16#0;
   STAT3[405] := B#16#0;
   STAT3[406] := B#16#0;
   STAT3[407] := B#16#0;
   STAT3[408] := B#16#0;
   STAT3[409] := B#16#0;
   STAT3[410] := B#16#0;
   STAT3[411] := B#16#0;
   STAT3[412] := B#16#0;
   STAT3[413] := B#16#0;
   STAT3[414] := B#16#0;
   STAT3[415] := B#16#0;
   STAT3[416] := B#16#0;
   STAT3[417] := B#16#0;
   STAT3[418] := B#16#0;
   STAT3[419] := B#16#0;
   STAT3[420] := B#16#0;
   STAT3[421] := B#16#0;
   STAT3[422] := B#16#0;
   STAT3[423] := B#16#0;
   STAT3[424] := B#16#0;
   STAT3[425] := B#16#0;
   STAT3[426] := B#16#0;
   STAT3[427] := B#16#0;
   STAT3[428] := B#16#0;
   STAT3[429] := B#16#0;
   STAT3[430] := B#16#0;
   STAT3[431] := B#16#0;
   STAT3[432] := B#16#0;
   STAT3[433] := B#16#0;
   STAT3[434] := B#16#0;
   STAT3[435] := B#16#0;
   STAT3[436] := B#16#0;
   STAT3[437] := B#16#0;
   STAT3[438] := B#16#0;
   STAT3[439] := B#16#0;
   STAT3[440] := B#16#0;
   STAT3[441] := B#16#0;
   STAT3[442] := B#16#0;
   STAT3[443] := B#16#0;
   STAT3[444] := B#16#0;
   STAT3[445] := B#16#0;
   STAT3[446] := B#16#0;
   STAT3[447] := B#16#0;
   STAT3[448] := B#16#0;
   STAT3[449] := B#16#0;
   STAT3[450] := B#16#0;
   STAT3[451] := B#16#0;
   STAT3[452] := B#16#0;
   STAT3[453] := B#16#0;
   STAT3[454] := B#16#0;
   STAT3[455] := B#16#0;
   STAT3[456] := B#16#0;
   STAT3[457] := B#16#0;
   STAT3[458] := B#16#0;
   STAT3[459] := B#16#0;
   STAT3[460] := B#16#0;
   STAT3[461] := B#16#0;
   STAT3[462] := B#16#0;
   STAT3[463] := B#16#0;
   STAT3[464] := B#16#0;
   STAT3[465] := B#16#0;
   STAT3[466] := B#16#0;
   STAT3[467] := B#16#0;
   STAT3[468] := B#16#0;
   STAT3[469] := B#16#0;
   STAT3[470] := B#16#0;
   STAT3[471] := B#16#0;
   STAT3[472] := B#16#0;
   STAT3[473] := B#16#0;
   STAT3[474] := B#16#0;
   STAT3[475] := B#16#0;
   STAT3[476] := B#16#0;
   STAT3[477] := B#16#0;
   STAT3[478] := B#16#0;
   STAT3[479] := B#16#0;
   STAT3[480] := B#16#0;
   STAT3[481] := B#16#0;
   STAT3[482] := B#16#0;
   STAT3[483] := B#16#0;
   STAT3[484] := B#16#0;
   STAT3[485] := B#16#0;
   STAT3[486] := B#16#0;
   STAT3[487] := B#16#0;
   STAT3[488] := B#16#0;
   STAT3[489] := B#16#0;
   STAT3[490] := B#16#0;
   STAT3[491] := B#16#0;
   STAT3[492] := B#16#0;
   STAT3[493] := B#16#0;
   STAT3[494] := B#16#0;
   STAT3[495] := B#16#0;
   STAT3[496] := B#16#0;
   STAT3[497] := B#16#0;
   STAT3[498] := B#16#0;
   STAT3[499] := B#16#0;
   STAT3[500] := B#16#0;
   STAT3[501] := B#16#0;
   STAT3[502] := B#16#0;
   STAT3[503] := B#16#0;
   STAT3[504] := B#16#0;
   STAT3[505] := B#16#0;
   STAT3[506] := B#16#0;
   STAT3[507] := B#16#0;
   STAT3[508] := B#16#0;
   STAT3[509] := B#16#0;
   STAT3[510] := B#16#0;
   STAT3[511] := B#16#0;
   STAT3[512] := B#16#0;
   STAT4 := '6ES7 318-3EL01-0AB0 ';
   STAT5[1] := B#16#3;
   STAT5[2] := B#16#2;
   STAT5[3] := B#16#B;
   STAT6 := W#16#0;
   STAT7[1] := W#16#1;
   STAT7[2] := W#16#1;
   STAT7[3] := W#16#0;
   STAT7[4] := W#16#0;
   STAT7[5] := W#16#0;
   STAT7[6] := W#16#0;
   STAT7[7] := W#16#0;
   STAT7[8] := W#16#0;
   STAT7[9] := W#16#0;
   STAT7[10] := W#16#0;
   STAT7[11] := W#16#0;
   STAT7[12] := W#16#0;
   STAT7[13] := W#16#0;
   STAT7[14] := W#16#0;
   STAT7[15] := W#16#0;
   STAT7[16] := W#16#0;
   STAT7[17] := W#16#0;
   STAT7[18] := W#16#0;
   STAT7[19] := W#16#0;
   STAT7[20] := W#16#0;
   STAT7[21] := W#16#0;
   STAT7[22] := W#16#0;
   STAT7[23] := W#16#0;
   STAT7[24] := W#16#0;
   STAT7[25] := W#16#0;
   STAT7[26] := W#16#0;
   STAT7[27] := W#16#0;
   STAT7[28] := W#16#0;
   STAT7[29] := W#16#0;
   STAT7[30] := W#16#0;
   STAT7[31] := W#16#0;
   STAT7[32] := W#16#0;
   STAT7[33] := W#16#1;
   STAT7[34] := W#16#0;
   STAT7[35] := W#16#0;
   STAT7[36] := W#16#0;
   STAT7[37] := W#16#0;
   STAT7[38] := W#16#0;
   STAT7[39] := W#16#0;
   STAT7[40] := W#16#0;
   STAT7[41] := W#16#0;
   STAT7[42] := W#16#0;
   STAT7[43] := W#16#0;
   STAT7[44] := W#16#0;
   STAT7[45] := W#16#0;
   STAT7[46] := W#16#0;
   STAT7[47] := W#16#0;
   STAT7[48] := W#16#0;
   STAT8 := FALSE;
   STAT9 := FALSE;
   STAT10 := FALSE;
   STAT11 := 0;
   STAT12 := 0;
   STAT13 := 2048;
   STAT14 := W#16#0;
   STAT15 := 0;
   STAT16 := 0;
   STAT17 := 0;
   STAT18 := 0;
   STAT19 := 0;
   STAT20 := 0;
   STAT21 := 0;
   STAT22 := 0;
   STAT23 := 0;
   STAT24 := W#16#0;
   STAT25 := FALSE;
   STAT26 := FALSE;
   STAT27 := FALSE;
   STAT28 := W#16#0;
   STAT29 := 0;
   STAT30 := 0;
   STAT31 := FALSE;
   STAT32 := FALSE;
   STAT33 := FALSE;
   STAT34 := FALSE;
   STAT35 := FALSE;
   STAT36 := FALSE;
   STAT37 := FALSE;
   STAT38 := FALSE;
   STAT39 := FALSE;
   STAT40 := FALSE;
   STAT41 := FALSE;
   STAT42 := W#16#0;
   STAT43 := 0;
   STAT44 := DW#16#80000000;
   STAT45 := 0;
   STAT46 := W#16#0;
   STAT47 := 'Device-MLFB';
   STAT48 := W#16#0;
   STAT49[0] := W#16#1;
   STAT49[1] := W#16#2;
   STAT49[2] := W#16#64;
   STAT49[3] := W#16#0;
   STAT49[4] := W#16#0;
   STAT49[5] := W#16#0;
   STAT49[6] := W#16#0;
   STAT49[7] := W#16#0;
   STAT49[8] := W#16#0;
   STAT49[9] := W#16#0;
   STAT49[10] := W#16#0;
   STAT49[11] := W#16#0;
   STAT49[12] := W#16#0;
   STAT49[13] := W#16#0;
   STAT49[14] := W#16#0;
   STAT49[15] := W#16#0;
   STAT49[16] := W#16#0;
   STAT49[17] := W#16#0;
   STAT49[18] := W#16#0;
   STAT49[19] := W#16#0;
   STAT49[20] := W#16#0;
   STAT49[21] := W#16#0;
   STAT49[22] := W#16#0;
   STAT49[23] := W#16#0;
   STAT49[24] := W#16#0;
   STAT49[25] := W#16#0;
   STAT49[26] := W#16#0;
   STAT49[27] := W#16#0;
   STAT49[28] := W#16#0;
   STAT49[29] := W#16#0;
   STAT49[30] := W#16#0;
   STAT49[31] := W#16#0;
   STAT49[32] := W#16#0;
   STAT49[33] := W#16#0;
   STAT49[34] := W#16#0;
   STAT49[35] := W#16#0;
   STAT49[36] := W#16#0;
   STAT49[37] := W#16#0;
   STAT49[38] := W#16#0;
   STAT49[39] := W#16#0;
   STAT49[40] := W#16#0;
   STAT49[41] := W#16#0;
   STAT49[42] := W#16#0;
   STAT49[43] := W#16#0;
   STAT49[44] := W#16#0;
   STAT49[45] := W#16#0;
   STAT49[46] := W#16#0;
   STAT49[47] := W#16#0;
   STAT50 := 3;
   STAT51 := DW#16#0;
   STAT52 := W#16#64;
   STAT53 := W#16#147;
   STAT54 := W#16#9C2;
   STAT55 := W#16#111;
   STAT56 := W#16#1FC9;
   STAT57 := W#16#1;
   STAT58 := W#16#692;
   STAT59 := W#16#1;
   STAT60 := W#16#1;
   STAT61 := W#16#0;
   STAT62 := 0;
   STAT63 := 0;
   STAT64 := 0;
   STAT65 := 0;
   STAT66 := 0;
   STAT67 := 512;
   STAT68 := 17671;
   STAT69 := 0;
   STAT70 := 0;
   STAT71 := 4;
   STAT72 := 0;
   STAT73 := 1;
   STAT74 := 326;
   STAT75 := 0;
   STAT76 := 2;
   STAT77 := 0;
   STAT78 := 0;
   STAT79 := 0;
   STAT80 := 0;
   STAT81 := 33;
   STAT82 := 0;
   STAT83 := 0;
   STAT84 := 2498;
   STAT85 := 2048;
   STAT86 := 0;
   STAT87 := 0;
   STAT88 := 257;
   STAT89 := 0;
   STAT90 := 14;
   STAT91 := 0;
   STAT92 := 0;
   STAT93 := 0;
   STAT94 := 0;
   STAT95 := B#16#0;
   STAT96 := B#16#3;
   STAT97 := B#16#4;
   STAT98 := B#16#0;
   STAT99[0] := B#16#0;
   STAT99[1] := B#16#0;
   STAT99[2] := B#16#0;
   STAT99[3] := B#16#0;
   STAT99[4] := B#16#0;
   STAT99[5] := B#16#0;
   STAT99[6] := B#16#0;
   STAT99[7] := B#16#0;
   STAT99[8] := B#16#0;
   STAT99[9] := B#16#0;
   STAT99[10] := B#16#0;
   STAT99[11] := B#16#0;
   STAT99[12] := B#16#0;
   STAT99[13] := B#16#0;
   STAT99[14] := B#16#0;
   STAT99[15] := B#16#0;
   STAT99[16] := B#16#0;
   STAT99[17] := B#16#0;
   STAT99[18] := B#16#0;
   STAT99[19] := B#16#0;
   STAT99[20] := B#16#0;
   STAT99[21] := B#16#0;
   STAT99[22] := B#16#0;
   STAT99[23] := B#16#0;
   STAT99[24] := B#16#0;
   STAT99[25] := B#16#0;
   STAT99[26] := B#16#0;
   STAT99[27] := B#16#0;
   STAT99[28] := B#16#0;
   STAT99[29] := B#16#0;
   STAT99[30] := B#16#0;
   STAT99[31] := B#16#0;
   STAT99[32] := B#16#0;
   STAT99[33] := B#16#0;
   STAT99[34] := B#16#0;
   STAT99[35] := B#16#0;
   STAT99[36] := B#16#0;
   STAT99[37] := B#16#0;
   STAT99[38] := B#16#0;
   STAT99[39] := B#16#0;
   STAT99[40] := B#16#0;
   STAT99[41] := B#16#0;
   STAT99[42] := B#16#0;
   STAT99[43] := B#16#0;
   STAT99[44] := B#16#0;
   STAT99[45] := B#16#0;
   STAT99[46] := B#16#0;
   STAT99[47] := B#16#0;
   STAT100 := FALSE;
   STAT101 := FALSE;
   STAT102 := FALSE;
   STAT103 := TRUE;
   STAT104 := FALSE;
   STAT105 := FALSE;
   STAT106 := FALSE;
   STAT107 := FALSE;
   STAT108 := FALSE;
   STAT109 := FALSE;
   STAT110 := FALSE;
   STAT111 := FALSE;
   STAT112 := FALSE;
   STAT113 := FALSE;
   STAT114 := FALSE;
   STAT115[1] := W#16#94;
   STAT115[2] := W#16#294;
   STAT115[3] := W#16#694;
   STAT115[4] := W#16#794;
   STAT116[1] := W#16#4094;
   STAT116[2] := W#16#4294;
   STAT116[3] := W#16#4694;
   STAT116[4] := W#16#794;
   STAT117[1] := W#16#92;
   STAT117[2] := W#16#292;
   STAT117[3] := W#16#692;
   STAT118[1] := W#16#4092;
   STAT118[2] := W#16#4292;
   STAT118[3] := W#16#4692;
   STAT119[1] := 0;
   STAT119[2] := 0;
   STAT119[3] := 0;
   STAT119[4] := 0;
   STAT119[5] := 0;
   STAT119[6] := 0;
   STAT119[7] := 0;
   STAT119[8] := 0;
   STAT119[9] := 0;
   STAT119[10] := 0;
   STAT120.REQ := FALSE;
   STAT120.ID := DW#16#0;
   STAT120.INDEX := 0;
   STAT120.MLEN := 0;
   STAT120.VALID := FALSE;
   STAT120.BUSY := FALSE;
   STAT120.ERROR := FALSE;
   STAT120.STATUS := DW#16#0;
   STAT120.LEN := 0;
   STAT131.MODE := 1;
   STAT131.F_ID := DW#16#1FFE;
   STAT131.MLEN := 28;
   STAT131.NEW := TRUE;
   STAT131.STATUS := DW#16#0;
   STAT131.ID := DW#16#1FC9;
   STAT131.LEN := 0;
   STAT131.TINFO := P#DB326.DBX 2196.0 BYTE 26;
   STAT131.AINFO := P#DB326.DBX 2168.0 BYTE 28;
   STAT141.STAT142 := W#16#102;
   STAT141.STAT143 := W#16#1;
   STAT144.STAT145 := B#16#13;
   STAT144.STAT146 := B#16#82;
   STAT144.STAT147 := B#16#1B;
   STAT144.STAT148 := B#16#64;
   STAT144.STAT149 := B#16#C7;
   STAT144.STAT150 := B#16#72;
   STAT144.STAT151 := W#16#494E;
   STAT144.STAT152 := DW#16#8107710;
   STAT153 := DW#16#100;
   STAT154 := W#16#1FC9;
   STAT155 := W#16#1;
   STAT156 := W#16#101;
   STAT157 := W#16#0;
   STAT158 := 14;
   STAT159 := 26;
   STAT160 := 0;
   STAT161 := 0;
   STAT162 := 1;
   STAT163 := 0;
   STAT164 := 2;
   STAT165 := B#16#54;
   STAT166 := FALSE;
   STAT167[1] := B#16#90;
   STAT167[2] := B#16#1;
   STAT167[3] := B#16#1;
   STAT167[4] := B#16#0;
   STAT167[5] := B#16#0;
   STAT167[6] := B#16#0;
   STAT167[7] := B#16#0;
   STAT167[8] := B#16#2;
   STAT167[9] := B#16#0;
   STAT167[10] := B#16#0;
   STAT167[11] := B#16#0;
   STAT167[12] := B#16#0;
   STAT167[13] := B#16#0;
   STAT167[14] := B#16#0;
   STAT167[15] := B#16#0;
   STAT167[16] := B#16#0;
   STAT168[0] := B#16#A;
   STAT168[1] := B#16#1;
   STAT168[2] := B#16#0;
   STAT168[3] := B#16#2;
   STAT168[4] := B#16#0;
   STAT168[5] := B#16#C;
   STAT168[6] := B#16#0;
   STAT168[7] := B#16#2;
   STAT168[8] := B#16#80;
   STAT168[9] := B#16#D6;
   STAT168[10] := B#16#42;
   STAT168[11] := B#16#0;
   STAT168[12] := B#16#13;
   STAT168[13] := B#16#A0;
   STAT168[14] := B#16#0;
   STAT168[15] := B#16#0;
   STAT168[16] := B#16#20;
   STAT168[17] := B#16#40;
   STAT168[18] := B#16#FF;
   STAT168[19] := B#16#FF;
   STAT168[20] := B#16#FF;
   STAT168[21] := B#16#FF;
   STAT168[22] := B#16#FF;
   STAT168[23] := B#16#FF;
   STAT168[24] := B#16#FF;
   STAT168[25] := B#16#FF;
   STAT168[26] := B#16#FF;
   STAT168[27] := B#16#0;
   STAT169[0] := B#16#38;
   STAT169[1] := B#16#C4;
   STAT169[2] := B#16#1A;
   STAT169[3] := B#16#56;
   STAT169[4] := B#16#C0;
   STAT169[5] := B#16#54;
   STAT169[6] := B#16#1F;
   STAT169[7] := B#16#FE;
   STAT169[8] := B#16#1F;
   STAT169[9] := B#16#C9;
   STAT169[10] := B#16#1;
   STAT169[11] := B#16#E;
   STAT169[12] := B#16#15;
   STAT169[13] := B#16#9;
   STAT169[14] := B#16#25;
   STAT169[15] := B#16#15;
   STAT169[16] := B#16#25;
   STAT169[17] := B#16#54;
   STAT169[18] := B#16#18;
   STAT169[19] := B#16#26;
   STAT169[20] := B#16#1;
   STAT169[21] := B#16#E;
   STAT169[22] := B#16#0;
   STAT169[23] := B#16#1;
   STAT169[24] := B#16#0;
   STAT169[25] := B#16#0;
   STAT170 := T#0MS;
   STAT171 := T#0MS;
   STAT172 := FALSE;
   STAT173 := FALSE;
   STAT174 := FALSE;
   STAT175 := FALSE;
   STAT176 := FALSE;
   STAT177 := FALSE;
   STAT178 := FALSE;
   STAT179 := FALSE;
   STAT180[2] := B#16#0;
   STAT180[3] := B#16#0;
   STAT180[4] := B#16#0;
   STAT180[5] := B#16#0;
   STAT180[6] := B#16#0;
   STAT180[7] := B#16#0;
   STAT180[8] := B#16#0;
   STAT180[9] := B#16#0;
   STAT180[10] := B#16#0;
   STAT180[11] := B#16#0;
   STAT180[12] := B#16#0;
   STAT180[13] := B#16#0;
   STAT180[14] := B#16#0;
   STAT180[15] := B#16#0;
   STAT180[16] := B#16#0;
   STAT180[17] := B#16#0;
   STAT180[18] := B#16#0;
   STAT180[19] := B#16#0;
   STAT180[20] := B#16#0;
   STAT181[0] := B#16#2;
   STAT181[1] := B#16#2;
   STAT181[2] := B#16#0;
   STAT181[3] := B#16#0;
   STAT181[4] := B#16#0;
   STAT181[5] := B#16#0;
   STAT181[6] := B#16#0;
   STAT181[7] := B#16#0;
   STAT181[8] := B#16#0;
   STAT181[9] := B#16#0;
   STAT181[10] := B#16#0;
   STAT181[11] := B#16#0;
   STAT181[12] := B#16#0;
   STAT181[13] := B#16#0;
   STAT181[14] := B#16#0;
   STAT181[15] := B#16#0;
   STAT181[16] := B#16#0;
   STAT181[17] := B#16#0;
   STAT181[18] := B#16#0;
   STAT181[19] := B#16#0;
   STAT181[20] := B#16#0;
   STAT181[21] := B#16#0;
   STAT181[22] := B#16#0;
   STAT181[23] := B#16#0;
   STAT181[24] := B#16#0;
   STAT181[25] := B#16#0;
   STAT181[26] := B#16#0;
   STAT181[27] := B#16#0;
   STAT181[28] := B#16#0;
   STAT181[29] := B#16#0;
   STAT181[30] := B#16#0;
   STAT181[31] := B#16#0;
   STAT181[32] := B#16#0;
   STAT181[33] := B#16#0;
   STAT181[34] := B#16#0;
   STAT181[35] := B#16#0;
   STAT181[36] := B#16#0;
   STAT181[37] := B#16#0;
   STAT181[38] := B#16#0;
   STAT181[39] := B#16#0;
   STAT181[40] := B#16#0;
   STAT181[41] := B#16#0;
   STAT181[42] := B#16#0;
   STAT181[43] := B#16#0;
   STAT181[44] := B#16#0;
   STAT181[45] := B#16#0;
   STAT181[46] := B#16#0;
   STAT181[47] := B#16#0;
   STAT182[1] := B#16#1;
   STAT182[2] := B#16#51;
   STAT183 := '';
   STAT184 := '';
   STAT185 := '';
   STAT186 := '';
   STAT187[0] := 7;
   STAT187[1] := -20496;
   STAT187[2] := -20495;
   STAT187[3] := -20494;
   STAT187[4] := -20493;
   STAT187[5] := -8180;
   STAT187[6] := -8190;
   STAT187[7] := -1983;
   STAT188[1] := B#16#0;
   STAT188[2] := B#16#0;
   STAT188[3] := B#16#0;
   STAT188[4] := B#16#0;
   STAT188[5] := B#16#0;
   STAT188[6] := B#16#0;
   STAT189[1] := B#16#0;
   STAT189[2] := B#16#0;
   STAT189[3] := B#16#0;
   STAT189[4] := B#16#0;
   STAT190[1] := B#16#0;
   STAT190[2] := B#16#0;
   STAT190[3] := B#16#0;
   STAT190[4] := B#16#0;
   STAT191[1] := B#16#0;
   STAT191[2] := B#16#0;
   STAT191[3] := B#16#0;
   STAT191[4] := B#16#0;
   STAT192 := '';
   STAT193 := 0;
   STAT194 := 0;
END_DATA_BLOCK

ORGANIZATION_BLOCK OB 1
TITLE =
VERSION : 0.1


VAR_TEMP
  TEMP0 : BYTE ;
  TEMP1 : BYTE ;
  TEMP2 : BYTE ;
  TEMP3 : BYTE ;
  TEMP4 : BYTE ;
  TEMP5 : BYTE ;
  TEMP6 : INT ;
  TEMP7 : INT ;
  TEMP8 : INT ;
  TEMP9 : DATE_AND_TIME ;
END_VAR
BEGIN
NETWORK
TITLE =

      AN    OV;
      =     M      3.3;
NETWORK
TITLE =

      A     OV;
      =     M      3.2;
      =     M     99.7;
NETWORK
TITLE =
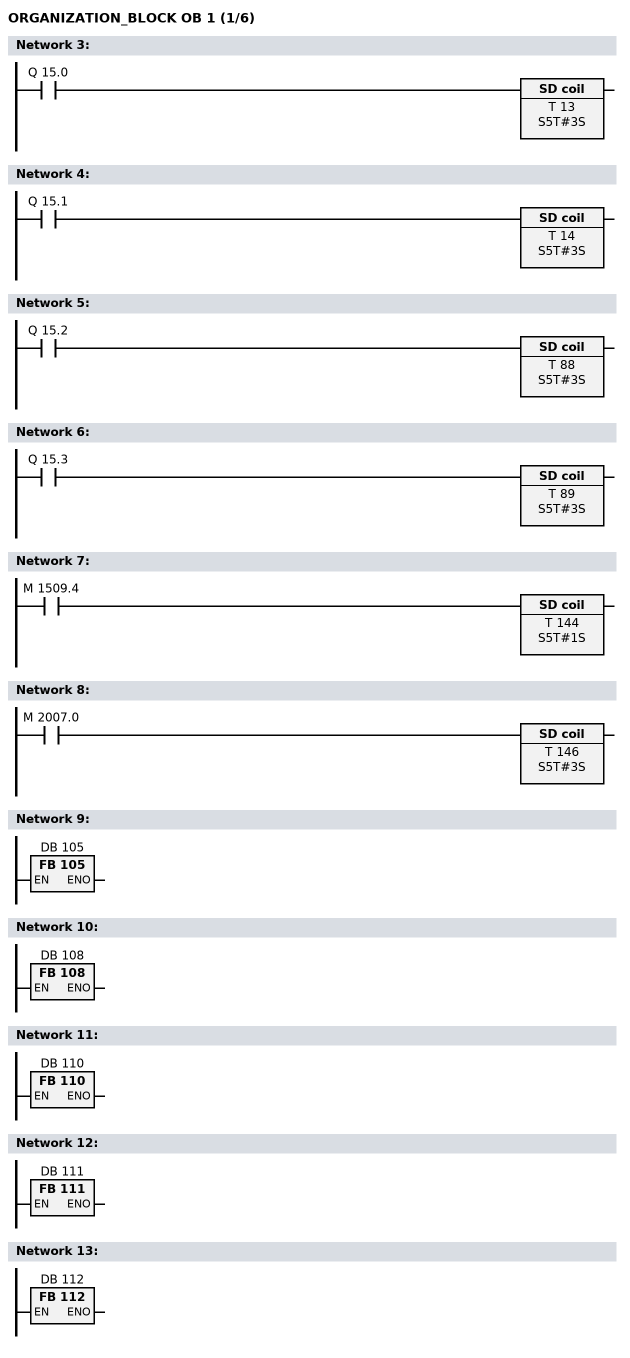

      A     Q     15.0;
      L     S5T#3S;
      SD    T     13;
NETWORK
TITLE =

      A     Q     15.1;
      L     S5T#3S;
      SD    T     14;
NETWORK
TITLE =

      A     Q     15.2;
      L     S5T#3S;
      SD    T     88;
NETWORK
TITLE =

      A     Q     15.3;
      L     S5T#3S;
      SD    T     89;
NETWORK
TITLE =

      A     M   1509.4;
      L     S5T#1S;
      SD    T    144;
NETWORK
TITLE =

      A     M   2007.0;
      L     S5T#3S;
      SD    T    146;
NETWORK
TITLE =

      CALL FB   105 , DB   105 ;
      NOP   0;
NETWORK
TITLE =

      CALL FB   108 , DB   108 ;
      NOP   0;
NETWORK
TITLE =

      CALL FB   110 , DB   110 ;
      NOP   0;
NETWORK
TITLE =

      CALL FB   111 , DB   111 ;
      NOP   0;
NETWORK
TITLE =

      CALL FB   112 , DB   112 ;
      NOP   0;
NETWORK
TITLE =
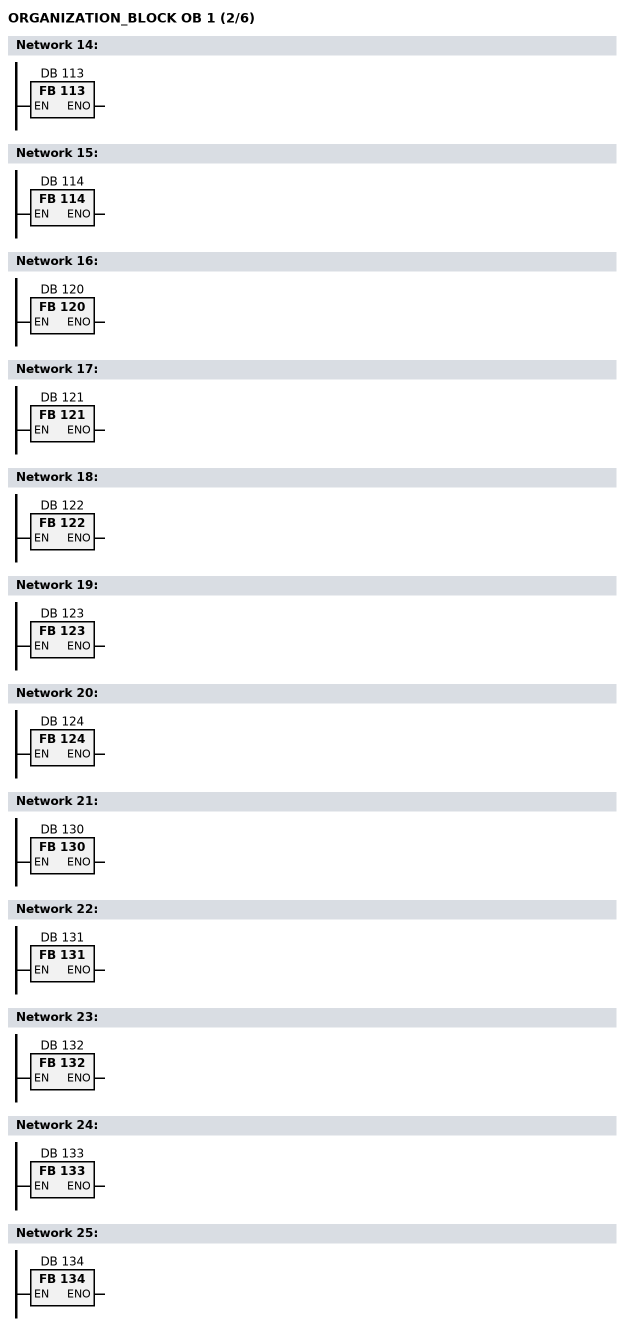

      CALL FB   113 , DB   113 ;
      NOP   0;
NETWORK
TITLE =

      CALL FB   114 , DB   114 ;
      NOP   0;
NETWORK
TITLE =

      CALL FB   120 , DB   120 ;
      NOP   0;
NETWORK
TITLE =

      CALL FB   121 , DB   121 ;
      NOP   0;
NETWORK
TITLE =

      CALL FB   122 , DB   122 ;
      NOP   0;
NETWORK
TITLE =

      CALL FB   123 , DB   123 ;
      NOP   0;
NETWORK
TITLE =

      CALL FB   124 , DB   124 ;
      NOP   0;
NETWORK
TITLE =

      CALL FB   130 , DB   130 ;
      NOP   0;
NETWORK
TITLE =

      CALL FB   131 , DB   131 ;
      NOP   0;
NETWORK
TITLE =

      CALL FB   132 , DB   132 ;
      NOP   0;
NETWORK
TITLE =

      CALL FB   133 , DB   133 ;
      NOP   0;
NETWORK
TITLE =

      CALL FB   134 , DB   134 ;
      NOP   0;
NETWORK
TITLE =
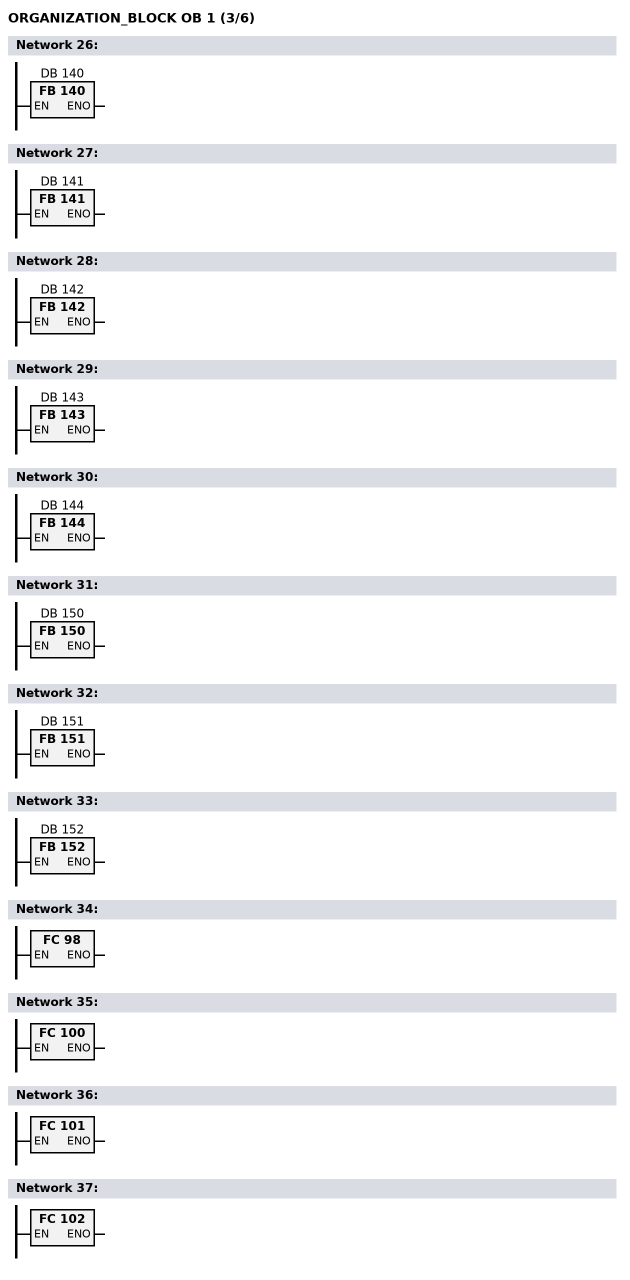

      CALL FB   140 , DB   140 ;
      NOP   0;
NETWORK
TITLE =

      CALL FB   141 , DB   141 ;
      NOP   0;
NETWORK
TITLE =

      CALL FB   142 , DB   142 ;
      NOP   0;
NETWORK
TITLE =

      CALL FB   143 , DB   143 ;
      NOP   0;
NETWORK
TITLE =

      CALL FB   144 , DB   144 ;
      NOP   0;
NETWORK
TITLE =

      CALL FB   150 , DB   150 ;
      NOP   0;
NETWORK
TITLE =

      CALL FB   151 , DB   151 ;
      NOP   0;
NETWORK
TITLE =

      CALL FB   152 , DB   152 ;
      NOP   0;
NETWORK
TITLE =

      CALL FC    98 ;
      NOP   0;
NETWORK
TITLE =

      CALL FC   100 ;
      NOP   0;
NETWORK
TITLE =

      CALL FC   101 ;
      NOP   0;
NETWORK
TITLE =

      CALL FC   102 ;
      NOP   0;
NETWORK
TITLE =
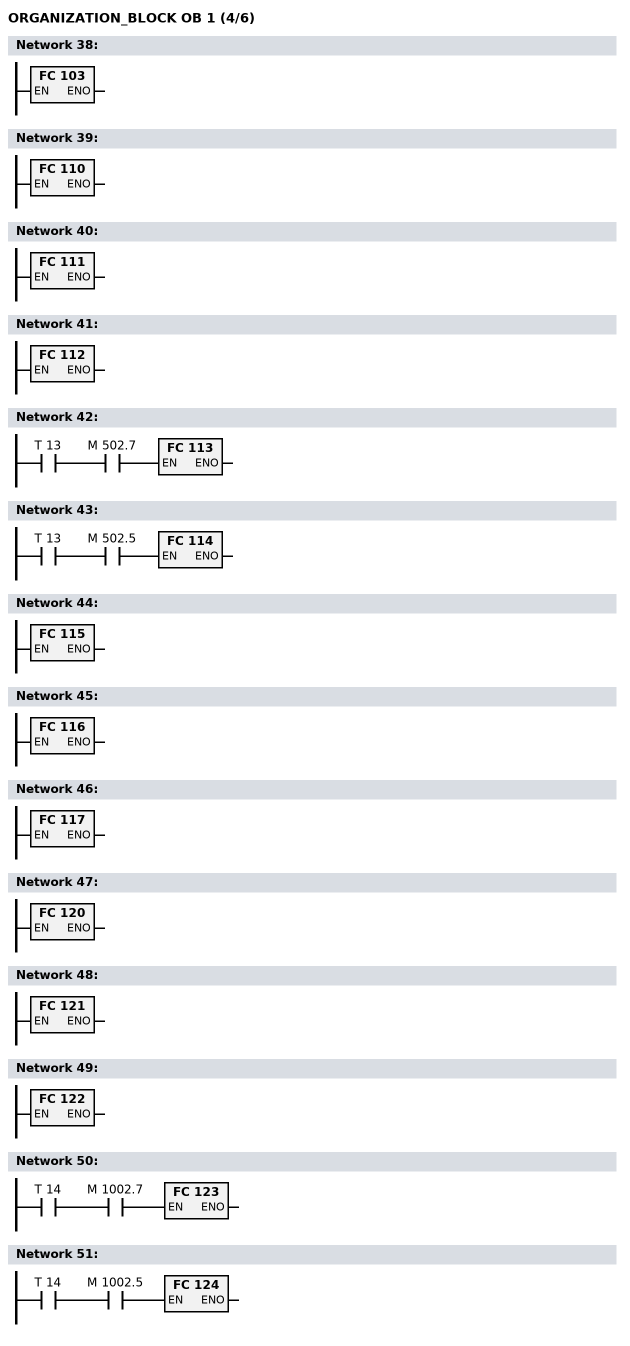

      CALL FC   103 ;
      NOP   0;
NETWORK
TITLE =

      CALL FC   110 ;
      NOP   0;
NETWORK
TITLE =

      CALL FC   111 ;
      NOP   0;
NETWORK
TITLE =

      CALL FC   112 ;
      NOP   0;
NETWORK
TITLE =

      A     T     13;
      A     M    502.7;
      JNB   _001;
      CALL FC   113 ;
_001: NOP   0;
NETWORK
TITLE =

      A     T     13;
      A     M    502.5;
      JNB   _002;
      CALL FC   114 ;
_002: NOP   0;
NETWORK
TITLE =

      CALL FC   115 ;
      NOP   0;
NETWORK
TITLE =

      CALL FC   116 ;
      NOP   0;
NETWORK
TITLE =

      CALL FC   117 ;
      NOP   0;
NETWORK
TITLE =

      CALL FC   120 ;
      NOP   0;
NETWORK
TITLE =

      CALL FC   121 ;
      NOP   0;
NETWORK
TITLE =

      CALL FC   122 ;
      NOP   0;
NETWORK
TITLE =

      A     T     14;
      A     M   1002.7;
      JNB   _003;
      CALL FC   123 ;
_003: NOP   0;
NETWORK
TITLE =

      A     T     14;
      A     M   1002.5;
      JNB   _004;
      CALL FC   124 ;
_004: NOP   0;
NETWORK
TITLE =
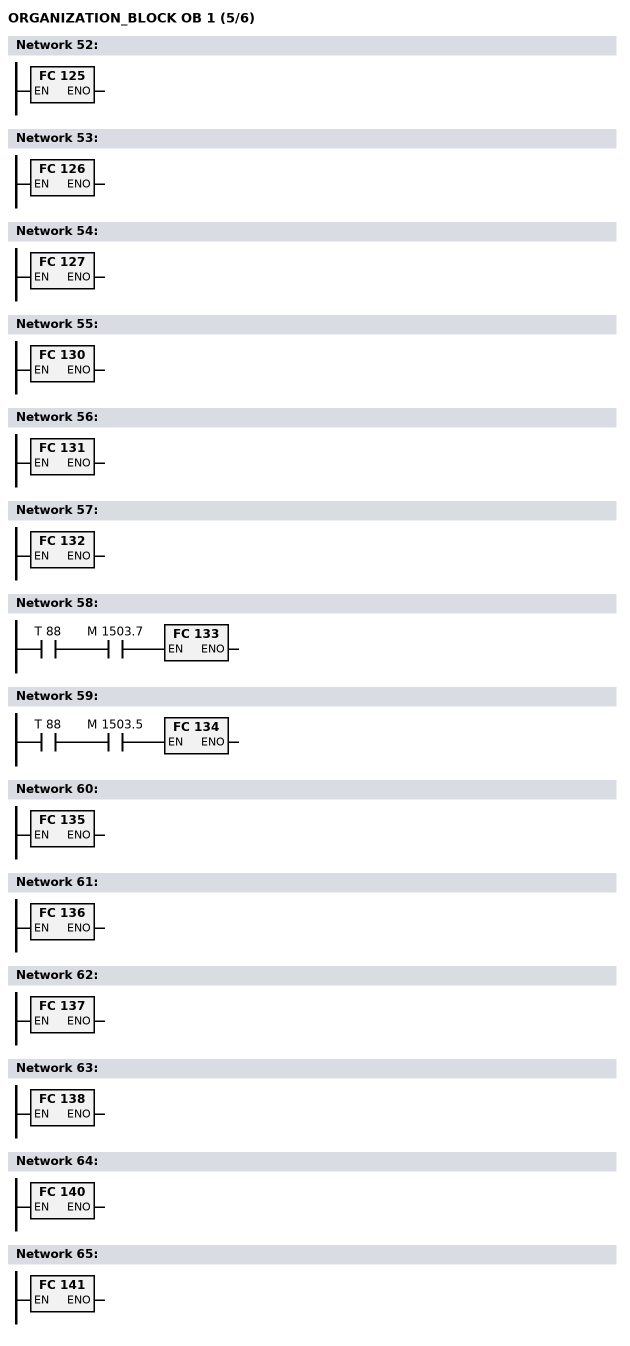

      CALL FC   125 ;
      NOP   0;
NETWORK
TITLE =

      CALL FC   126 ;
      NOP   0;
NETWORK
TITLE =

      CALL FC   127 ;
      NOP   0;
NETWORK
TITLE =

      CALL FC   130 ;
      NOP   0;
NETWORK
TITLE =

      CALL FC   131 ;
      NOP   0;
NETWORK
TITLE =

      CALL FC   132 ;
      NOP   0;
NETWORK
TITLE =

      A     T     88;
      A     M   1503.7;
      JNB   _005;
      CALL FC   133 ;
_005: NOP   0;
NETWORK
TITLE =

      A     T     88;
      A     M   1503.5;
      JNB   _006;
      CALL FC   134 ;
_006: NOP   0;
NETWORK
TITLE =

      CALL FC   135 ;
      NOP   0;
NETWORK
TITLE =

      CALL FC   136 ;
      NOP   0;
NETWORK
TITLE =

      CALL FC   137 ;
      NOP   0;
NETWORK
TITLE =

      CALL FC   138 ;
      NOP   0;
NETWORK
TITLE =

      CALL FC   140 ;
      NOP   0;
NETWORK
TITLE =

      CALL FC   141 ;
      NOP   0;
NETWORK
TITLE =
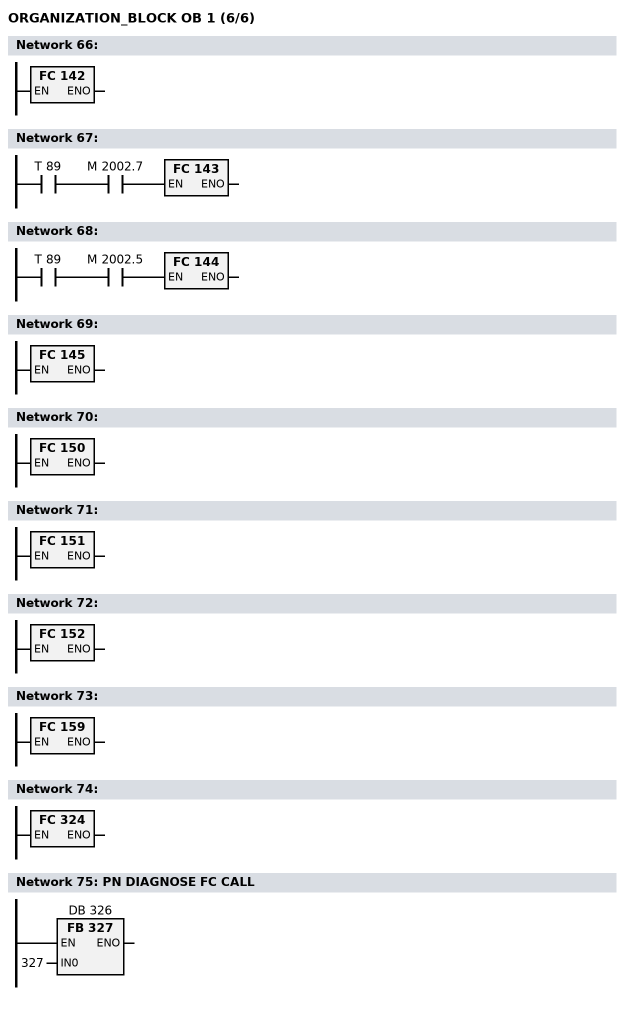

      CALL FC   142 ;
      NOP   0;
NETWORK
TITLE =

      A     T     89;
      A     M   2002.7;
      JNB   _007;
      CALL FC   143 ;
_007: NOP   0;
NETWORK
TITLE =

      A     T     89;
      A     M   2002.5;
      JNB   _008;
      CALL FC   144 ;
_008: NOP   0;
NETWORK
TITLE =

      CALL FC   145 ;
      NOP   0;
NETWORK
TITLE =

      CALL FC   150 ;
      NOP   0;
NETWORK
TITLE =

      CALL FC   151 ;
      NOP   0;
NETWORK
TITLE =

      CALL FC   152 ;
      NOP   0;
NETWORK
TITLE =

      CALL FC   159 ;
      NOP   0;
NETWORK
TITLE =

      CALL FC   324 ;
      NOP   0;
NETWORK
TITLE =PN DIAGNOSE FC CALL

      CALL FB   327 , DB   326 (
           IN0                      := 327);

      NOP   0;
END_ORGANIZATION_BLOCK

ORGANIZATION_BLOCK OB 80
TITLE = "Cycle Time Fault"
VERSION : 0.1


VAR_TEMP
  OB80_EV_CLASS : BYTE ;	//16#35, Event class 3, Entering event state, Internal fault event
  OB80_FLT_ID : BYTE ;	//16#XX, Fault identifcation code
  OB80_PRIORITY : BYTE ;	//Priority of OB Execution
  OB80_OB_NUMBR : BYTE ;	//80 (Organization block 80, OB80)
  OB80_RESERVED_1 : BYTE ;	//Reserved for system
  OB80_RESERVED_2 : BYTE ;	//Reserved for system
  OB80_ERROR_INFO : WORD ;	//Error information on event
  OB80_ERR_EV_CLASS : BYTE ;	//Class of event causing error
  OB80_ERR_EV_NUM : BYTE ;	//Number of event causing error
  OB80_OB_PRIORITY : BYTE ;	//Priority of OB causing error
  OB80_OB_NUM : BYTE ;	//Number of OB causing error
  OB80_DATE_TIME : DATE_AND_TIME ;	//Date and time OB80 started
END_VAR
BEGIN
NETWORK
TITLE =

END_ORGANIZATION_BLOCK

ORGANIZATION_BLOCK OB 82
TITLE = "I/O Point Fault"
VERSION : 0.1


VAR_TEMP
  OB82_EV_CLASS : BYTE ;	//16#39, Event class 3, Entering event state, Internal fault event
  OB82_FLT_ID : BYTE ;	//16#XX, Fault identifcation code
  OB82_PRIORITY : BYTE ;	//Priority of OB Execution
  OB82_OB_NUMBR : BYTE ;	//82 (Organization block 82, OB82)
  OB82_RESERVED_1 : BYTE ;	//Reserved for system
  OB82_IO_FLAG : BYTE ;	//Input (01010100), Output (01010101)
  OB82_MDL_ADDR : WORD ;	//Base address of module with fault
  OB82_MDL_DEFECT : BOOL ;	//Module defective
  OB82_INT_FAULT : BOOL ;	//Internal fault
  OB82_EXT_FAULT : BOOL ;	//External fault
  OB82_PNT_INFO : BOOL ;	//Point information
  OB82_EXT_VOLTAGE : BOOL ;	//External voltage low
  OB82_FLD_CONNCTR : BOOL ;	//Field wiring connector missing
  OB82_NO_CONFIG : BOOL ;	//Module has no configuration data
  OB82_CONFIG_ERR : BOOL ;	//Module has configuration error
  OB82_MDL_TYPE : BYTE ;	//Type of module
  OB82_SUB_MDL_ERR : BOOL ;	//Sub-Module is missing or has error
  OB82_COMM_FAULT : BOOL ;	//Communication fault
  OB82_MDL_STOP : BOOL ;	//Module is stopped
  OB82_WTCH_DOG_FLT : BOOL ;	//Watch dog timer stopped module
  OB82_INT_PS_FLT : BOOL ;	//Internal power supply fault
  OB82_PRIM_BATT_FLT : BOOL ;	//Primary battery is in fault
  OB82_BCKUP_BATT_FLT : BOOL ;	//Backup battery is in fault
  OB82_RESERVED_2 : BOOL ;	//Reserved for system
  OB82_RACK_FLT : BOOL ;	//Rack fault, only for bus interface module
  OB82_PROC_FLT : BOOL ;	//Processor fault
  OB82_EPROM_FLT : BOOL ;	//EPROM fault
  OB82_RAM_FLT : BOOL ;	//RAM fault
  OB82_ADU_FLT : BOOL ;	//ADU fault
  OB82_FUSE_FLT : BOOL ;	//Fuse fault
  OB82_HW_INTR_FLT : BOOL ;	//Hardware interupt input in fault
  OB82_RESERVED_3 : BOOL ;	//Reserved for system
  OB82_DATE_TIME : DATE_AND_TIME ;	//Date and time OB82 started
END_VAR
BEGIN
NETWORK
TITLE =PN DIAGNOSE FC CALL

      CALL FB   327 , DB   326 (
           IN0                      := 327);

      NOP   0;
NETWORK
TITLE = Call report System Error Block

END_ORGANIZATION_BLOCK

ORGANIZATION_BLOCK OB 83
TITLE = "I/O Point Fault"
VERSION : 0.1


VAR_TEMP
  OB83_EV_CLASS : BYTE ;	//16#38/39, Event class 3, module inserted/removed (8/9)
  OB83_FLT_ID : BYTE ;	//16#XX, Fault identifcation code
  OB83_PRIORITY : BYTE ;	//Priority of OB Execution
  OB83_OB_NUMBR : BYTE ;	//83 (Organization block 83, OB83)
  OB83_RESERVED_1 : BYTE ;	//Reserved for system
  OB83_MDL_ID : BYTE ;	//Input module (01010100), Output module (01010101)
  OB83_MDL_ADDR : WORD ;	//Base address of module with point fault
  OB83_RACK_NUM : INT ;	//Number of rack that has module with point fault
  OB83_MDL_TYPE : WORD ;	//Module type with point fault
  OB83_DATE_TIME : DATE_AND_TIME ;	//Date and time OB83 started
END_VAR
BEGIN
NETWORK
TITLE =PN DIAGNOSE FC CALL

      CALL FB   327 , DB   326 (
           IN0                      := 327);

      NOP   0;
NETWORK
TITLE = Call report System Error Block

END_ORGANIZATION_BLOCK

ORGANIZATION_BLOCK OB 85
TITLE = "Organization Block (OB) Not Loaded Fault"
VERSION : 0.1


VAR_TEMP
  OB85_EV_CLASS : BYTE ;	//16#35 Event class 3
  OB85_FLT_ID : BYTE ;	//16#XX, Fault identification code
  OB85_PRIORITY : BYTE ;	//Priority of OB Execution
  OB85_OB_NUMBR : BYTE ;	//85 (Organization block 85, OB85)
  OB85_RESERVED_1 : BYTE ;	//Reserved for system
  OB85_RESERVED_2 : BYTE ;	//Reserved for system
  OB85_RESERVED_3 : INT ;	//Reserved for system
  OB85_ERR_EV_CLASS : BYTE ;	//Class of event causing error
  OB85_ERR_EV_NUM : BYTE ;	//Number of event causing error
  OB85_OB_PRIOR : BYTE ;	//Priority of OB causing error
  OB85_OB_NUM : BYTE ;	//Number of OB causing error
  OB85_DATE_TIME : DATE_AND_TIME ;	//Date and time OB85 started
END_VAR
BEGIN
NETWORK
TITLE =

END_ORGANIZATION_BLOCK

ORGANIZATION_BLOCK OB 86
TITLE = "Loss Of Rack Fault"
VERSION : 0.1


VAR_TEMP
  OB86_EV_CLASS : BYTE ;	//16#38/39 Event class 3
  OB86_FLT_ID : BYTE ;	//16#C1/C4/C5, Fault identifcation code
  OB86_PRIORITY : BYTE ;	//Priority of OB Execution
  OB86_OB_NUMBR : BYTE ;	//86 (Organization block 86, OB86)
  OB86_RESERVED_1 : BYTE ;	//Reserved for system
  OB86_RESERVED_2 : BYTE ;	//Reserved for system
  OB86_MDL_ADDR : WORD ;	//Base address of IM module in rack with fault
  OB86_RACKS_FLTD : ARRAY  [0 .. 31 ] OF BOOL ;	//Racks in fault
  OB86_DATE_TIME : DATE_AND_TIME ;	//Date and time OB86 started
END_VAR
BEGIN
NETWORK
TITLE =PN DIAGNOSE FC CALL

      CALL FB   327 , DB   326 (
           IN0                      := 327);

      NOP   0;
NETWORK
TITLE = Call report System Error Block

END_ORGANIZATION_BLOCK

ORGANIZATION_BLOCK OB 87
TITLE = "Communication Fault"
VERSION : 0.1


VAR_TEMP
  OB87_EV_CLASS : BYTE ;	//16#39 Event class 3
  OB87_FLT_ID : BYTE ;	//16#XX, Fault identifcation code
  OB87_PRIORITY : BYTE ;	//Priority of OB Execution
  OB87_OB_NUMBR : BYTE ;	//87 (Organization block 87, OB87)
  OB87_RESERVED_1 : BYTE ;	//Reserved for system
  OB87_RESERVED_2 : BYTE ;	//Reserved for system
  OB87_RESERVED_3 : WORD ;	//Reserved for system
  OB87_RESERVED_4 : DWORD ;	//Reserved for system
  OB87_DATE_TIME : DATE_AND_TIME ;	//Date and time OB87 started
END_VAR
BEGIN
NETWORK
TITLE =

END_ORGANIZATION_BLOCK

ORGANIZATION_BLOCK OB 100
TITLE = "Complete Restart"
VERSION : 0.1


VAR_TEMP
  OB100_EV_CLASS : BYTE ;	//16#13, Event class 1, Entering event state, Event logged in diagnostic buffer
  OB100_STRTUP : BYTE ;	//16#81/82/83/84 Method of startup
  OB100_PRIORITY : BYTE ;	//Priority of OB Execution
  OB100_OB_NUMBR : BYTE ;	//100 (Organization block 100, OB100)
  OB100_RESERVED_1 : BYTE ;	//Reserved for system
  OB100_RESERVED_2 : BYTE ;	//Reserved for system
  OB100_STOP : WORD ;	//Event that caused CPU to stop (16#4xxx)
  OB100_STRT_INFO : DWORD ;	//Information on how system started
  OB100_DATE_TIME : DATE_AND_TIME ;	//Date and time OB100 started
END_VAR
BEGIN
NETWORK
TITLE =PN DIAGNOSE FC CALL

      CALL FB   327 , DB   326 (
           IN0                      := 327);

      NOP   0;
END_ORGANIZATION_BLOCK

ORGANIZATION_BLOCK OB 121
TITLE = "Programming Error"
VERSION : 0.1


VAR_TEMP
  OB121_EV_CLASS : BYTE ;	//16#25, Event class 2, Entering event state, Internal fault event
  OB121_SW_FLT : BYTE ;	//16#XX Software programming fault
  OB121_PRIORITY : BYTE ;	//Priority of OB Execution
  OB121_OB_NUMBR : BYTE ;	//121 (Organization block 121, OB121)
  OB121_BLK_TYPE : BYTE ;	//16#88/8A/8B/8C/8E Type of block fault occured in
  OB121_RESERVED_1 : BYTE ;	//Reserved for system
  OB121_FLT_REG : WORD ;	//16#XX Specific register that caused fault
  OB121_BLK_NUM : WORD ;	//Number of block that programming fault occured in
  OB121_PRG_ADDR : WORD ;	//Address in block where programming fault occured
  OB121_DATE_TIME : DATE_AND_TIME ;	//Date and time OB121 started
END_VAR
BEGIN
NETWORK
TITLE =

END_ORGANIZATION_BLOCK

ORGANIZATION_BLOCK OB 122
TITLE = "Module Access Error"
VERSION : 0.1


VAR_TEMP
  OB122_EV_CLASS : BYTE ;	//16#29, Event class 2, Entering event state, Internal fault event
  OB122_SW_FLT : BYTE ;	//16#XX Software error code
  OB122_PRIORITY : BYTE ;	//Priority of OB Execution
  OB122_OB_NUMBR : BYTE ;	//122 (Organization block 122, OB122)
  OB122_BLK_TYPE : BYTE ;	//16#88/8C/8E Type of block fault occured in
  OB122_MEM_AREA : BYTE ;	//Memory area where access error occured
  OB122_MEM_ADDR : WORD ;	//Memory address where access error occured
  OB122_BLK_NUM : WORD ;	//Block number in which error occured
  OB122_PRG_ADDR : WORD ;	//Program address where error occured
  OB122_DATE_TIME : DATE_AND_TIME ;	//Date and time OB1 started
END_VAR
BEGIN
NETWORK
TITLE =

END_ORGANIZATION_BLOCK

